   W_o[8,37] := 0.2716717;
   W_o[8,38] := -0.5921684;
   W_o[8,39] := 0.1613293;
   W_o[9,0] := -0.6345086;
   W_o[9,1] := -0.259372;
   W_o[9,2] := -0.4410478;
   W_o[9,3] := -0.1479532;
   W_o[9,4] := 0.07470662;
   W_o[9,5] := -0.1442392;
   W_o[9,6] := 0.2044672;
   W_o[9,7] := -0.3629733;
   W_o[9,8] := -0.8357224;
   W_o[9,9] := -0.03687909;
   W_o[9,10] := -0.5277801;
   W_o[9,11] := 0.1395604;
   W_o[9,12] := 0.00705423;
   W_o[9,13] := -0.06065191;
   W_o[9,14] := 0.00270301;
   W_o[9,15] := 0.02473978;
   W_o[9,16] := -0.1366292;
   W_o[9,17] := -0.1191437;
   W_o[9,18] := -0.06459489;
   W_o[9,19] := -0.155962;
   W_o[9,20] := -0.1332201;
   W_o[9,21] := 0.6168138;
   W_o[9,22] := -0.008209;
   W_o[9,23] := -0.03221058;
   W_o[9,24] := -0.07914114;
   W_o[9,25] := -0.2822376;
   W_o[9,26] := 0.1799158;
   W_o[9,27] := 0.1354283;
   W_o[9,28] := 0.1905717;
   W_o[9,29] := 0.3257442;
   W_o[9,30] := 0.2045423;
   W_o[9,31] := 0.117547;
   W_o[9,32] := 0.1869259;
   W_o[9,33] := 0.4169515;
   W_o[9,34] := 0.131826;
   W_o[9,35] := -0.1867882;
   W_o[9,36] := -0.09728058;
   W_o[9,37] := -0.2151765;
   W_o[9,38] := 0.03850761;
   W_o[9,39] := -0.0044641;
   W_o[10,0] := 0.06105608;
   W_o[10,1] := -0.06832715;
   W_o[10,2] := 0.07474305;
   W_o[10,3] := -0.08913961;
   W_o[10,4] := -0.2327598;
   W_o[10,5] := 0.07582341;
   W_o[10,6] := 0.104368;
   W_o[10,7] := 0.03688281;
   W_o[10,8] := -0.01102509;
   W_o[10,9] := -0.02805536;
   W_o[10,10] := 0.1092547;
   W_o[10,11] := -0.04491638;
   W_o[10,12] := -0.00955069;
   W_o[10,13] := -0.3600228;
   W_o[10,14] := -0.2598117;
   W_o[10,15] := -0.1312952;
   W_o[10,16] := 0.1270282;
   W_o[10,17] := 0.2455932;
   W_o[10,18] := 0.02347365;
   W_o[10,19] := 0.08953306;
   W_o[10,20] := -0.412829;
   W_o[10,21] := -0.1269261;
   W_o[10,22] := 0.1430949;
   W_o[10,23] := -0.2883692;
   W_o[10,24] := 1.613103;
   W_o[10,25] := 1.56905;
   W_o[10,26] := 0.11707;
   W_o[10,27] := -0.6253218;
   W_o[10,28] := -0.570655;
   W_o[10,29] := 0.06348585;
   W_o[10,30] := 0.2199306;
   W_o[10,31] := -0.02762064;
   W_o[10,32] := 0.08508236;
   W_o[10,33] := 0.2603731;
   W_o[10,34] := 0.5238683;
   W_o[10,35] := -0.3072915;
   W_o[10,36] := 0.4589803;
   W_o[10,37] := -0.3261147;
   W_o[10,38] := -0.04951124;
   W_o[10,39] := -0.0165583;
   W_o[11,0] := 0.2717895;
   W_o[11,1] := 0.4973186;
   W_o[11,2] := -0.111147;
   W_o[11,3] := 0.00516717;
   W_o[11,4] := -0.7287747;
   W_o[11,5] := -0.07876529;
   W_o[11,6] := -0.5072603;
   W_o[11,7] := -0.03536538;
   W_o[11,8] := 0.1201321;
   W_o[11,9] := 0.1112787;
   W_o[11,10] := 0.1532365;
   W_o[11,11] := -0.4891608;
   W_o[11,12] := 0.1887655;
   W_o[11,13] := 0.1852349;
   W_o[11,14] := 0.1703349;
   W_o[11,15] := -0.2467272;
   W_o[11,16] := 0.04845995;
   W_o[11,17] := 0.2819173;
   W_o[11,18] := 0.1057306;
   W_o[11,19] := -0.00306271;
   W_o[11,20] := -0.724054;
   W_o[11,21] := 0.09254762;
   W_o[11,22] := -0.4099866;
   W_o[11,23] := -0.1073627;
   W_o[11,24] := -0.0586772;
   W_o[11,25] := 0.3430104;
   W_o[11,26] := 0.1855343;
   W_o[11,27] := 0.1084731;
   W_o[11,28] := 0.5040212;
   W_o[11,29] := -0.00853192;
   W_o[11,30] := -0.3662441;
   W_o[11,31] := -0.01966033;
   W_o[11,32] := -0.06275205;
   W_o[11,33] := 0.09751767;
   W_o[11,34] := -0.2004695;
   W_o[11,35] := -0.1034404;
   W_o[11,36] := 0.2302412;
   W_o[11,37] := 0.1414506;
   W_o[11,38] := 0.266502;
   W_o[11,39] := -0.3097887;
   W_o[12,0] := -0.01830707;
   W_o[12,1] := 0.131161;
   W_o[12,2] := 0.00496979;
   W_o[12,3] := 0.2061931;
   W_o[12,4] := 0.03057155;
   W_o[12,5] := 0.02297443;
   W_o[12,6] := 0.05931674;
   W_o[12,7] := -0.03210922;
   W_o[12,8] := 0.07573608;
   W_o[12,9] := 0.1248056;
   W_o[12,10] := -0.07253183;
   W_o[12,11] := -0.2442229;
   W_o[12,12] := 0.1326389;
   W_o[12,13] := -0.1664325;
   W_o[12,14] := -0.1405273;
   W_o[12,15] := -0.05658006;
   W_o[12,16] := 0.04406866;
   W_o[12,17] := 0.0236842;
   W_o[12,18] := 0.7910394;
   W_o[12,19] := 0.02559086;
   W_o[12,20] := -0.1635535;
   W_o[12,21] := -0.01013497;
   W_o[12,22] := -0.3506611;
   W_o[12,23] := -0.1885774;
   W_o[12,24] := 0.4997112;
   W_o[12,25] := 0.5154855;
   W_o[12,26] := 0.1843938;
   W_o[12,27] := 0.02656424;
   W_o[12,28] := 0.00674596;
   W_o[12,29] := 0.03458697;
   W_o[12,30] := -0.4318717;
   W_o[12,31] := -0.1312484;
   W_o[12,32] := -0.3812101;
   W_o[12,33] := -0.02800291;
   W_o[12,34] := -0.2285903;
   W_o[12,35] := 0.123769;
   W_o[12,36] := 0.08067092;
   W_o[12,37] := -0.04127869;
   W_o[12,38] := -0.06010977;
   W_o[12,39] := -0.00181283;
   W_o[13,0] := -0.04045204;
   W_o[13,1] := -0.3968439;
   W_o[13,2] := 0.08165251;
   W_o[13,3] := -0.01278869;
   W_o[13,4] := -0.4479226;
   W_o[13,5] := -0.2656083;
   W_o[13,6] := 0.3235124;
   W_o[13,7] := 0.574206;
   W_o[13,8] := -0.2794143;
   W_o[13,9] := 0.3598377;
   W_o[13,10] := -0.08126416;
   W_o[13,11] := -0.00919488;
   W_o[13,12] := 0.09122144;
   W_o[13,13] := 0.02155786;
   W_o[13,14] := 0.1209246;
   W_o[13,15] := -0.00289959;
   W_o[13,16] := -0.2549352;
   W_o[13,17] := -0.2486969;
   W_o[13,18] := 0.6917394;
   W_o[13,19] := -0.03206153;
   W_o[13,20] := -0.2219304;
   W_o[13,21] := 0.1183459;
   W_o[13,22] := 0.3679306;
   W_o[13,23] := 0.4413242;
   W_o[13,24] := 1.975207;
   W_o[13,25] := 1.843769;
   W_o[13,26] := -0.279261;
   W_o[13,27] := -0.3077843;
   W_o[13,28] := -0.01960251;
   W_o[13,29] := -0.2369677;
   W_o[13,30] := 0.109645;
   W_o[13,31] := -0.1079782;
   W_o[13,32] := 0.038799;
   W_o[13,33] := 0.05485996;
   W_o[13,34] := 0.5972548;
   W_o[13,35] := 0.01886969;
   W_o[13,36] := 0.09835773;
   W_o[13,37] := 0.3843534;
   W_o[13,38] := 0.05617079;
   W_o[13,39] := -0.2227704;
   W_o[14,0] := 0.8289077;
   W_o[14,1] := -0.2031105;
   W_o[14,2] := 0.03403382;
   W_o[14,3] := 0.05452057;
   W_o[14,4] := 0.2272833;
   W_o[14,5] := -0.07046781;
   W_o[14,6] := 0.3896516;
   W_o[14,7] := 0.4871905;
   W_o[14,8] := -0.07724485;
   W_o[14,9] := -0.07247894;
   W_o[14,10] := 0.2814783;
   W_o[14,11] := -0.02350411;
   W_o[14,12] := 0.3741138;
   W_o[14,13] := 0.01457606;
   W_o[14,14] := -0.08907567;
   W_o[14,15] := 0.03109477;
   W_o[14,16] := 0.05151353;
   W_o[14,17] := -0.1566754;
   W_o[14,18] := -0.2640311;
   W_o[14,19] := -0.1076154;
   W_o[14,20] := 0.3854151;
   W_o[14,21] := 1.575822;
   W_o[14,22] := -0.05344179;
   W_o[14,23] := -0.9402446;
   W_o[14,24] := -0.0189026;
   W_o[14,25] := -0.00721721;
   W_o[14,26] := -0.4206359;
   W_o[14,27] := 0.5079048;
   W_o[14,28] := 0.2300513;
   W_o[14,29] := 0.2341685;
   W_o[14,30] := -0.1072616;
   W_o[14,31] := -0.05015407;
   W_o[14,32] := 0.03626099;
   W_o[14,33] := 0.2209553;
   W_o[14,34] := 0.2829649;
   W_o[14,35] := -0.102007;
   W_o[14,36] := 0.00415739;
   W_o[14,37] := 0.2021578;
   W_o[14,38] := 0.1449325;
   W_o[14,39] := 0.1953939;
   W_o[15,0] := 0.00236452;
   W_o[15,1] := 0.6316325;
   W_o[15,2] := 0.04516845;
   W_o[15,3] := -0.1972448;
   W_o[15,4] := -0.6675987;
   W_o[15,5] := 0.3806524;
   W_o[15,6] := 0.6475521;
   W_o[15,7] := 0.2695197;
   W_o[15,8] := -0.4985425;
   W_o[15,9] := -0.3775528;
   W_o[15,10] := 0.255392;
   W_o[15,11] := -0.1499313;
   W_o[15,12] := 0.5755351;
   W_o[15,13] := -0.03951031;
   W_o[15,14] := 0.02471058;
   W_o[15,15] := -0.2347889;
   W_o[15,16] := 0.3119133;
   W_o[15,17] := 0.02724188;
   W_o[15,18] := 0.3374691;
   W_o[15,19] := -0.0329643;
   W_o[15,20] := -0.8862573;
   W_o[15,21] := 0.5019892;
   W_o[15,22] := -0.01491885;
   W_o[15,23] := 0.393534;
   W_o[15,24] := 0.2951014;
   W_o[15,25] := 0.4423684;
   W_o[15,26] := -0.03397221;
   W_o[15,27] := -0.4513796;
   W_o[15,28] := 0.261473;
   W_o[15,29] := -0.1054694;
   W_o[15,30] := 0.3078526;
   W_o[15,31] := -0.1044204;
   W_o[15,32] := 0.2778185;
   W_o[15,33] := -0.00624027;
   W_o[15,34] := 0.2965292;
   W_o[15,35] := -0.2159247;
   W_o[15,36] := 0.05058118;
   W_o[15,37] := 0.00013962;
   W_o[15,38] := 1.000757;
   W_o[15,39] := 0.5571635;
   R_i[0,0] := -0.1137149;
   R_i[0,1] := -0.00305563;
   R_i[0,2] := 0.4498252;
   R_i[0,3] := 0.408096;
   R_i[0,4] := 0.4966823;
   R_i[0,5] := 0.2685225;
   R_i[0,6] := 0.5829936;
   R_i[0,7] := 0.309512;
   R_i[0,8] := 0.584756;
   R_i[0,9] := 0.4425567;
   R_i[0,10] := 0.168636;
   R_i[0,11] := -0.314454;
   R_i[0,12] := 0.01961905;
   R_i[0,13] := 0.3972826;
   R_i[0,14] := 0.3588874;
   R_i[0,15] := 0.1209446;
   R_i[1,0] := -0.03926941;
   R_i[1,1] := -0.2256729;
   R_i[1,2] := -0.1890858;
   R_i[1,3] := -0.4077013;
   R_i[1,4] := 1.580356;
   R_i[1,5] := -0.5334294;
   R_i[1,6] := -0.07024953;
   R_i[1,7] := 0.4276721;
   R_i[1,8] := -0.6611474;
   R_i[1,9] := 0.4677508;
   R_i[1,10] := -0.07782394;
   R_i[1,11] := -0.4426747;
   R_i[1,12] := 0.1923219;
   R_i[1,13] := 0.6306989;
   R_i[1,14] := -0.442345;
   R_i[1,15] := -0.1436543;
   R_i[2,0] := -0.1087616;
   R_i[2,1] := -0.00270978;
   R_i[2,2] := 0.2189552;
   R_i[2,3] := -0.5836519;
   R_i[2,4] := -0.07285596;
   R_i[2,5] := 0.04414057;
   R_i[2,6] := 0.2944021;
   R_i[2,7] := -0.5636789;
   R_i[2,8] := 0.02525483;
   R_i[2,9] := 0.2138523;
   R_i[2,10] := 0.1495301;
   R_i[2,11] := 0.4767698;
   R_i[2,12] := 0.3593693;
   R_i[2,13] := -0.475326;
   R_i[2,14] := -0.06119934;
   R_i[2,15] := -0.1814424;
   R_i[3,0] := -0.3477732;
   R_i[3,1] := -0.02923841;
   R_i[3,2] := -0.01545414;
   R_i[3,3] := 0.6730511;
   R_i[3,4] := 0.5243366;
   R_i[3,5] := 0.1240829;
   R_i[3,6] := 0.3667154;
   R_i[3,7] := 0.4002697;
   R_i[3,8] := 0.66468;
   R_i[3,9] := 0.1677333;
   R_i[3,10] := 0.1911234;
   R_i[3,11] := -0.5108734;
   R_i[3,12] := 0.1124746;
   R_i[3,13] := -0.2656624;
   R_i[3,14] := 0.3824491;
   R_i[3,15] := -0.1521915;
   R_i[4,0] := 0.00580328;
   R_i[4,1] := 0.6645847;
   R_i[4,2] := -0.7531157;
   R_i[4,3] := 0.00536597;
   R_i[4,4] := -1.547926;
   R_i[4,5] := -0.4703412;
   R_i[4,6] := -0.2358381;
   R_i[4,7] := 0.2062922;
   R_i[4,8] := 0.5056434;
   R_i[4,9] := 0.1705665;
   R_i[4,10] := -0.126984;
   R_i[4,11] := -1.014073;
   R_i[4,12] := 0.5201921;
   R_i[4,13] := -0.1478145;
   R_i[4,14] := -0.1872073;
   R_i[4,15] := -0.01908887;
   R_i[5,0] := -0.5724422;
   R_i[5,1] := 0.07744113;
   R_i[5,2] := 0.07027231;
   R_i[5,3] := 0.1578984;
   R_i[5,4] := 0.2315233;
   R_i[5,5] := 0.1378991;
   R_i[5,6] := -0.3647587;
   R_i[5,7] := -0.1986962;
   R_i[5,8] := -0.04011904;
   R_i[5,9] := -0.05832585;
   R_i[5,10] := -0.04800356;
   R_i[5,11] := -0.2021917;
   R_i[5,12] := -0.02367323;
   R_i[5,13] := 0.1801978;
   R_i[5,14] := 0.07786623;
   R_i[5,15] := -0.4144403;
   R_i[6,0] := -0.4898062;
   R_i[6,1] := -0.08807379;
   R_i[6,2] := 0.729624;
   R_i[6,3] := 0.5344335;
   R_i[6,4] := -0.3394561;
   R_i[6,5] := 0.02468326;
   R_i[6,6] := -0.5965754;
   R_i[6,7] := -0.1523064;
   R_i[6,8] := -0.06543954;
   R_i[6,9] := 0.0652044;
   R_i[6,10] := -0.09473334;
   R_i[6,11] := 0.06633532;
   R_i[6,12] := 0.5554917;
   R_i[6,13] := -0.5657542;
   R_i[6,14] := 0.1251685;
   R_i[6,15] := -1.210496;
   R_i[7,0] := 0.09141196;
   R_i[7,1] := -0.2953948;
   R_i[7,2] := -0.04736479;
   R_i[7,3] := 0.6381459;
   R_i[7,4] := -0.1735898;
   R_i[7,5] := 0.02200026;
   R_i[7,6] := -0.542483;
   R_i[7,7] := 0.4112348;
   R_i[7,8] := 0.08935327;
   R_i[7,9] := 0.211784;
   R_i[7,10] := 0.3778164;
   R_i[7,11] := -0.2455601;
   R_i[7,12] := -0.2529224;
   R_i[7,13] := 0.3676308;
   R_i[7,14] := -0.1642352;
   R_i[7,15] := 0.3013193;
   R_i[8,0] := -0.4359751;
   R_i[8,1] := 0.5370886;
   R_i[8,2] := -0.01918638;
   R_i[8,3] := 0.06577428;
   R_i[8,4] := -0.2360706;
   R_i[8,5] := 0.04361986;
   R_i[8,6] := 0.4372621;
   R_i[8,7] := 0.317978;
   R_i[8,8] := -1.000937;
   R_i[8,9] := -0.3358858;
   R_i[8,10] := 0.9401911;
   R_i[8,11] := -0.4844143;
   R_i[8,12] := -0.02272851;
   R_i[8,13] := 0.1828933;
   R_i[8,14] := -0.01882748;
   R_i[8,15] := -0.06172743;
   R_i[9,0] := -0.5143862;
   R_i[9,1] := 0.06295519;
   R_i[9,2] := 0.3046114;
   R_i[9,3] := 0.03788998;
   R_i[9,4] := 0.1308033;
   R_i[9,5] := -0.358474;
   R_i[9,6] := 0.69233;
   R_i[9,7] := -0.2776851;
   R_i[9,8] := 0.00155199;
   R_i[9,9] := -0.09497612;
   R_i[9,10] := 0.191216;
   R_i[9,11] := -0.428836;
   R_i[9,12] := 0.097583;
   R_i[9,13] := 0.2892125;
   R_i[9,14] := 0.1341387;
   R_i[9,15] := -0.6526389;
   R_i[10,0] := -1.243925;
   R_i[10,1] := 0.680451;
   R_i[10,2] := 0.9452817;
   R_i[10,3] := -1.115271;
   R_i[10,4] := -0.6274545;
   R_i[10,5] := -0.4702299;
   R_i[10,6] := 0.9055709;
   R_i[10,7] := 0.7863802;
   R_i[10,8] := 1.259396;
   R_i[10,9] := 0.4866133;
   R_i[10,10] := -0.232237;
   R_i[10,11] := -0.8811347;
   R_i[10,12] := -0.1416707;
   R_i[10,13] := 0.2519798;
   R_i[10,14] := 0.7145844;
   R_i[10,15] := -0.03913529;
   R_i[11,0] := -0.2986307;
   R_i[11,1] := 0.7416621;
   R_i[11,2] := -0.5418634;
   R_i[11,3] := -0.0208676;
   R_i[11,4] := 0.4454969;
   R_i[11,5] := -0.1592286;
   R_i[11,6] := 0.2505509;
   R_i[11,7] := -0.382692;
   R_i[11,8] := 0.1618413;
   R_i[11,9] := 0.4193928;
   R_i[11,10] := 0.02712804;
   R_i[11,11] := -1.186852;
   R_i[11,12] := 0.2001949;
   R_i[11,13] := 0.1532502;
   R_i[11,14] := -0.3284004;
   R_i[11,15] := -0.2820552;
   R_i[12,0] := -0.2895075;
   R_i[12,1] := 1.091435;
   R_i[12,2] := -0.05338987;
   R_i[12,3] := 0.2911161;
   R_i[12,4] := 0.1629717;
   R_i[12,5] := -0.161591;
   R_i[12,6] := 0.5146877;
   R_i[12,7] := 0.03626299;
   R_i[12,8] := 0.08357667;
   R_i[12,9] := 0.2767582;
   R_i[12,10] := -0.2725959;
   R_i[12,11] := -0.9445232;
   R_i[12,12] := 2.164176;
   R_i[12,13] := -0.04564672;
   R_i[12,14] := -0.9437686;
   R_i[12,15] := -0.3752556;
   R_i[13,0] := -0.3738814;
   R_i[13,1] := -0.4302073;
   R_i[13,2] := 0.06173271;
   R_i[13,3] := -0.3280604;
   R_i[13,4] := -0.2716264;
   R_i[13,5] := 0.3550667;
   R_i[13,6] := -0.05685175;
   R_i[13,7] := 0.5135436;
   R_i[13,8] := 0.1640313;
   R_i[13,9] := -0.2691319;
   R_i[13,10] := -0.3801848;
   R_i[13,11] := 0.1228051;
   R_i[13,12] := 0.5428029;
   R_i[13,13] := 1.709359;
   R_i[13,14] := 1.011569;
   R_i[13,15] := -0.4288203;
   R_i[14,0] := 0.2300761;
   R_i[14,1] := -1.012092;
   R_i[14,2] := 0.6361403;
   R_i[14,3] := 0.05786986;
   R_i[14,4] := -0.4553789;
   R_i[14,5] := -0.6679262;
   R_i[14,6] := -0.4034081;
   R_i[14,7] := 0.00973069;
   R_i[14,8] := 1.011842;
   R_i[14,9] := -0.3590509;
   R_i[14,10] := 0.3335861;
   R_i[14,11] := -0.8217174;
   R_i[14,12] := -0.6475059;
   R_i[14,13] := -0.2020338;
   R_i[14,14] := 3.036138;
   R_i[14,15] := -0.1744984;
   R_i[15,0] := -0.04125203;
   R_i[15,1] := 0.6700256;
   R_i[15,2] := 1.07735;
   R_i[15,3] := 0.2874972;
   R_i[15,4] := -0.03804383;
   R_i[15,5] := 0.0777116;
   R_i[15,6] := 0.6422315;
   R_i[15,7] := 0.2854839;
   R_i[15,8] := 0.2419276;
   R_i[15,9] := 0.0058566;
   R_i[15,10] := 0.6288991;
   R_i[15,11] := -0.8346034;
   R_i[15,12] := 0.2495139;
   R_i[15,13] := -0.4616964;
   R_i[15,14] := 0.8547717;
   R_i[15,15] := -1.059702;
   R_f[0,0] := 0.3233714;
   R_f[0,1] := -0.6415426;
   R_f[0,2] := 0.4436696;
   R_f[0,3] := -0.1691184;
   R_f[0,4] := -0.2260693;
   R_f[0,5] := 0.4070715;
   R_f[0,6] := 0.9958715;
   R_f[0,7] := -0.6152283;
   R_f[0,8] := -0.1669062;
   R_f[0,9] := 0.1140058;
   R_f[0,10] := -1.301264;
   R_f[0,11] := 0.6843588;
   R_f[0,12] := 0.2550505;
   R_f[0,13] := -0.5000576;
   R_f[0,14] := 1.899208;
   R_f[0,15] := 0.3119706;
   R_f[1,0] := -0.1011617;
   R_f[1,1] := 3.477333;
   R_f[1,2] := -0.2395845;
   R_f[1,3] := 0.2576158;
   R_f[1,4] := 0.6485823;
   R_f[1,5] := 0.2552066;
   R_f[1,6] := 0.4734288;
   R_f[1,7] := 0.4439468;
   R_f[1,8] := 0.08832169;
   R_f[1,9] := -0.07672439;
   R_f[1,10] := -0.1136505;
   R_f[1,11] := -0.1276775;
   R_f[1,12] := 0.153016;
   R_f[1,13] := 0.1081575;
   R_f[1,14] := -0.00451868;
   R_f[1,15] := 0.1695628;
   R_f[2,0] := 0.8806943;
   R_f[2,1] := -0.4307577;
   R_f[2,2] := -0.285418;
   R_f[2,3] := 0.7795734;
   R_f[2,4] := 0.49964;
   R_f[2,5] := 0.1542652;
   R_f[2,6] := 0.2286351;
   R_f[2,7] := -0.7402638;
   R_f[2,8] := -0.6850481;
   R_f[2,9] := -0.3444061;
   R_f[2,10] := -0.5146202;
   R_f[2,11] := 0.5203135;
   R_f[2,12] := -0.2921089;
   R_f[2,13] := -0.7581262;
   R_f[2,14] := 0.2400508;
   R_f[2,15] := 0.06470054;
   R_f[3,0] := -1.016384;
   R_f[3,1] := -0.01572494;
   R_f[3,2] := 1.122687;
   R_f[3,3] := -1.076523;
   R_f[3,4] := -0.2219028;
   R_f[3,5] := 0.3841916;
   R_f[3,6] := 0.6512823;
   R_f[3,7] := 1.68439;
   R_f[3,8] := 0.7787917;
   R_f[3,9] := -0.1303423;
   R_f[3,10] := 0.1025792;
   R_f[3,11] := 0.0630113;
   R_f[3,12] := -0.2613996;
   R_f[3,13] := 0.08574831;
   R_f[3,14] := 0.5817915;
   R_f[3,15] := -0.1694773;
   R_f[4,0] := -0.09817147;
   R_f[4,1] := -0.8673013;
   R_f[4,2] := 0.1123603;
   R_f[4,3] := -0.05304767;
   R_f[4,4] := -0.1617602;
   R_f[4,5] := -0.4315653;
   R_f[4,6] := -0.1545042;
   R_f[4,7] := -0.04651795;
   R_f[4,8] := -0.7793221;
   R_f[4,9] := 0.2078234;
   R_f[4,10] := 0.1676973;
   R_f[4,11] := 0.3325663;
   R_f[4,12] := 0.157971;
   R_f[4,13] := 0.7362291;
   R_f[4,14] := 0.0176266;
   R_f[4,15] := -0.6734453;
   R_f[5,0] := 1.169603;
   R_f[5,1] := -0.73158;
   R_f[5,2] := 0.4122632;
   R_f[5,3] := 0.02196453;
   R_f[5,4] := 0.3548708;
   R_f[5,5] := 0.1889586;
   R_f[5,6] := 0.3045126;
   R_f[5,7] := 0.9211732;
   R_f[5,8] := -0.4857724;
   R_f[5,9] := -0.9820208;
   R_f[5,10] := -0.5130315;
   R_f[5,11] := 0.2623543;
   R_f[5,12] := -0.2203466;
   R_f[5,13] := -1.837646;
   R_f[5,14] := -0.6587409;
   R_f[5,15] := -0.2930804;
   R_f[6,0] := -0.3989139;
   R_f[6,1] := -0.7530556;
   R_f[6,2] := 1.695848;
   R_f[6,3] := -0.1637086;
   R_f[6,4] := 0.2540572;
   R_f[6,5] := 0.02853256;
   R_f[6,6] := 0.1514727;
   R_f[6,7] := -1.134142;
   R_f[6,8] := -0.9914478;
   R_f[6,9] := -0.4490964;
   R_f[6,10] := -0.6475779;
   R_f[6,11] := -0.02062916;
   R_f[6,12] := 0.3351462;
   R_f[6,13] := 0.3090186;
   R_f[6,14] := 0.6139765;
   R_f[6,15] := 0.7687923;
   R_f[7,0] := -0.2705219;
   R_f[7,1] := 0.04162847;
   R_f[7,2] := 3.147241;
   R_f[7,3] := -0.331195;
   R_f[7,4] := -0.5884408;
   R_f[7,5] := -0.3636526;
   R_f[7,6] := -0.9163497;
   R_f[7,7] := 0.3539489;
   R_f[7,8] := 0.2825061;
   R_f[7,9] := 0.493275;
   R_f[7,10] := 1.353475;
   R_f[7,11] := -1.124487;
   R_f[7,12] := -0.5918967;
   R_f[7,13] := 1.290014;
   R_f[7,14] := -0.550961;
   R_f[7,15] := 0.8665411;
   R_f[8,0] := 0.3655965;
   R_f[8,1] := -1.387398;
   R_f[8,2] := 0.6403066;
   R_f[8,3] := 0.4521842;
   R_f[8,4] := 0.426568;
   R_f[8,5] := -0.3468258;
   R_f[8,6] := -1.100012;
   R_f[8,7] := -0.6693547;
   R_f[8,8] := -3.069017;
   R_f[8,9] := 0.1657671;
   R_f[8,10] := 0.784942;
   R_f[8,11] := -0.4345917;
   R_f[8,12] := -1.434882;
   R_f[8,13] := 0.1338141;
   R_f[8,14] := -0.793483;
   R_f[8,15] := -0.2249214;
   R_f[9,0] := -0.152597;
   R_f[9,1] := -1.499914;
   R_f[9,2] := 1.108761;
   R_f[9,3] := -0.5297781;
   R_f[9,4] := -0.6886869;
   R_f[9,5] := -1.672909;
   R_f[9,6] := 2.633435;
   R_f[9,7] := -1.828544;
   R_f[9,8] := -0.740662;
   R_f[9,9] := 1.526205;
   R_f[9,10] := 0.4746018;
   R_f[9,11] := 1.381489;
   R_f[9,12] := -0.6054185;
   R_f[9,13] := 0.7926679;
   R_f[9,14] := 0.3271781;
   R_f[9,15] := -1.000112;
   R_f[10,0] := 2.164407;
   R_f[10,1] := -0.6995372;
   R_f[10,2] := 0.6653332;
   R_f[10,3] := 1.181759;
   R_f[10,4] := -0.2965346;
   R_f[10,5] := -0.1037577;
   R_f[10,6] := 0.02757812;
   R_f[10,7] := -0.9681873;
   R_f[10,8] := -0.4607585;
   R_f[10,9] := -0.5446746;
   R_f[10,10] := 0.780597;
   R_f[10,11] := -0.7688502;
   R_f[10,12] := -1.056067;
   R_f[10,13] := -0.1988855;
   R_f[10,14] := 0.01456859;
   R_f[10,15] := 0.3702135;
   R_f[11,0] := 0.2434937;
   R_f[11,1] := -0.1798942;
   R_f[11,2] := 0.2355876;
   R_f[11,3] := -0.6682997;
   R_f[11,4] := -0.5007147;
   R_f[11,5] := -0.5791205;
   R_f[11,6] := 0.1253008;
   R_f[11,7] := -0.7620748;
   R_f[11,8] := -0.5787513;
   R_f[11,9] := 0.0264844;
   R_f[11,10] := 0.4317927;
   R_f[11,11] := -1.222577;
   R_f[11,12] := -0.03755289;
   R_f[11,13] := -0.1228497;
   R_f[11,14] := 0.0646783;
   R_f[11,15] := 0.2649987;
   R_f[12,0] := -0.02412502;
   R_f[12,1] := -0.4178893;
   R_f[12,2] := 0.2250565;
   R_f[12,3] := 0.2468531;
   R_f[12,4] := -0.2603359;
   R_f[12,5] := 0.5588626;
   R_f[12,6] := 0.3501927;
   R_f[12,7] := 0.0646469;
   R_f[12,8] := 0.3895332;
   R_f[12,9] := 0.409056;
   R_f[12,10] := 0.161415;
   R_f[12,11] := -0.05112006;
   R_f[12,12] := 1.493768;
   R_f[12,13] := 0.3131461;
   R_f[12,14] := 0.4573432;
   R_f[12,15] := 0.3800302;
   R_f[13,0] := 0.5914586;
   R_f[13,1] := -0.351166;
   R_f[13,2] := 0.8291268;
   R_f[13,3] := 0.2013447;
   R_f[13,4] := 0.82876;
   R_f[13,5] := 0.8977232;
   R_f[13,6] := 1.657781;
   R_f[13,7] := 0.4952854;
   R_f[13,8] := -0.8510268;
   R_f[13,9] := -0.7816306;
   R_f[13,10] := 0.3712052;
   R_f[13,11] := 0.7794952;
   R_f[13,12] := -0.1510022;
   R_f[13,13] := -0.1749281;
   R_f[13,14] := -0.00674355;
   R_f[13,15] := -0.6594451;
   R_f[14,0] := -0.03948923;
   R_f[14,1] := -0.3682528;
   R_f[14,2] := 1.244398;
   R_f[14,3] := -0.5374001;
   R_f[14,4] := -0.4286888;
   R_f[14,5] := 0.2608948;
   R_f[14,6] := 0.4886785;
   R_f[14,7] := 1.195282;
   R_f[14,8] := 0.1545673;
   R_f[14,9] := -1.140402;
   R_f[14,10] := 0.05182516;
   R_f[14,11] := -0.2172662;
   R_f[14,12] := 0.1702152;
   R_f[14,13] := -0.6474801;
   R_f[14,14] := 1.387721;
   R_f[14,15] := 0.2322865;
   R_f[15,0] := 0.3153065;
   R_f[15,1] := -0.9808237;
   R_f[15,2] := 0.2264991;
   R_f[15,3] := -0.2976737;
   R_f[15,4] := 0.5468484;
   R_f[15,5] := 0.7780918;
   R_f[15,6] := 2.003952;
   R_f[15,7] := 2.355743;
   R_f[15,8] := -0.1702361;
   R_f[15,9] := -0.381211;
   R_f[15,10] := 1.069254;
   R_f[15,11] := -0.3054578;
   R_f[15,12] := -0.4347287;
   R_f[15,13] := -1.114827;
   R_f[15,14] := 0.3245434;
   R_f[15,15] := -1.337709;
   R_g[0,0] := -2.805433;
   R_g[0,1] := 0.09675837;
   R_g[0,2] := 0.04763355;
   R_g[0,3] := 0.1613498;
   R_g[0,4] := -0.04916951;
   R_g[0,5] := 0.06786807;
   R_g[0,6] := 0.07195669;
   R_g[0,7] := 0.1879627;
   R_g[0,8] := 0.02096096;
   R_g[0,9] := -0.05091592;
   R_g[0,10] := 0.1711352;
   R_g[0,11] := 0.09710391;
   R_g[0,12] := -0.1928508;
   R_g[0,13] := 0.04608029;
   R_g[0,14] := 0.3775772;
   R_g[0,15] := -0.05004899;
   R_g[1,0] := 0.08712953;
   R_g[1,1] := -1.281738;
   R_g[1,2] := 0.486291;
   R_g[1,3] := -0.1018547;
   R_g[1,4] := 0.5911466;
   R_g[1,5] := 0.3826247;
   R_g[1,6] := 0.04029783;
   R_g[1,7] := 0.06582787;
   R_g[1,8] := -0.06752597;
   R_g[1,9] := -0.2294858;
   R_g[1,10] := -0.1253151;
   R_g[1,11] := -0.2067355;
   R_g[1,12] := -0.05208173;
   R_g[1,13] := 0.1810765;
   R_g[1,14] := 0.05905702;
   R_g[1,15] := -0.06634986;
   R_g[2,0] := -0.2549139;
   R_g[2,1] := -0.05303259;
   R_g[2,2] := -3.258265;
   R_g[2,3] := 0.2239036;
   R_g[2,4] := 0.08010214;
   R_g[2,5] := 0.1251935;
   R_g[2,6] := -0.1281362;
   R_g[2,7] := 0.03709217;
   R_g[2,8] := -0.0533942;
   R_g[2,9] := -0.1838315;
   R_g[2,10] := 0.01583981;
   R_g[2,11] := 0.1206139;
   R_g[2,12] := 0.02361463;
   R_g[2,13] := 0.1162473;
   R_g[2,14] := 0.1685608;
   R_g[2,15] := -0.04670952;
   R_g[3,0] := -0.3499806;
   R_g[3,1] := 0.7145555;
   R_g[3,2] := -0.7979932;
   R_g[3,3] := -2.84151;
   R_g[3,4] := 0.1580465;
   R_g[3,5] := -0.08033045;
   R_g[3,6] := -0.1452473;
   R_g[3,7] := 0.2225952;
   R_g[3,8] := 0.07427457;
   R_g[3,9] := 0.3725025;
   R_g[3,10] := -0.308892;
   R_g[3,11] := -0.2322429;
   R_g[3,12] := 0.6733903;
   R_g[3,13] := 0.1802014;
   R_g[3,14] := -0.04057474;
   R_g[3,15] := -0.1780594;
   R_g[4,0] := 0.4558564;
   R_g[4,1] := 0.2691017;
   R_g[4,2] := 0.2479934;
   R_g[4,3] := 0.1830495;
   R_g[4,4] := -2.643592;
   R_g[4,5] := -0.1854873;
   R_g[4,6] := 0.5796254;
   R_g[4,7] := -0.2360368;
   R_g[4,8] := 0.3996172;
   R_g[4,9] := -0.08552616;
   R_g[4,10] := -0.3547961;
   R_g[4,11] := 0.02176627;
   R_g[4,12] := -0.1695444;
   R_g[4,13] := -0.6054811;
   R_g[4,14] := 0.05480947;
   R_g[4,15] := 0.2614591;
   R_g[5,0] := 0.09851117;
   R_g[5,1] := 0.05978253;
   R_g[5,2] := -0.2238024;
   R_g[5,3] := 0.06287329;
   R_g[5,4] := 0.2952785;
   R_g[5,5] := -6.417284;
   R_g[5,6] := -0.01966351;
   R_g[5,7] := 0.08289347;
   R_g[5,8] := 0.2335418;
   R_g[5,9] := 0.4640638;
   R_g[5,10] := -0.5190796;
   R_g[5,11] := -0.3999299;
   R_g[5,12] := 0.3029557;
   R_g[5,13] := 0.06150499;
   R_g[5,14] := -1.054952;
   R_g[5,15] := -0.08431676;
   R_g[6,0] := -0.1025641;
   R_g[6,1] := 0.05051776;
   R_g[6,2] := 0.0306027;
   R_g[6,3] := 0.06608646;
   R_g[6,4] := -0.05028161;
   R_g[6,5] := -0.1038706;
   R_g[6,6] := -3.13754;
   R_g[6,7] := -0.1565541;
   R_g[6,8] := 0.03909466;
   R_g[6,9] := -0.03506904;
   R_g[6,10] := 0.0048442;
   R_g[6,11] := -0.1906409;
   R_g[6,12] := 0.330723;
   R_g[6,13] := -0.06755624;
   R_g[6,14] := -0.1569814;
   R_g[6,15] := -0.3220711;
   R_g[7,0] := 0.07863971;
   R_g[7,1] := -0.1875482;
   R_g[7,2] := -0.2537812;
   R_g[7,3] := -0.08824939;
   R_g[7,4] := -0.1294116;
   R_g[7,5] := 0.2885412;
   R_g[7,6] := 0.1121606;
   R_g[7,7] := -3.136752;
   R_g[7,8] := -0.08472223;
   R_g[7,9] := 0.00790842;
   R_g[7,10] := -0.1138648;
   R_g[7,11] := -0.05684523;
   R_g[7,12] := 0.1106585;
   R_g[7,13] := -0.07569506;
   R_g[7,14] := 0.4233017;
   R_g[7,15] := -0.1342552;
   R_g[8,0] := 0.08961181;
   R_g[8,1] := 0.4651947;
   R_g[8,2] := -0.3656231;
   R_g[8,3] := 0.2111352;
   R_g[8,4] := -0.00757714;
   R_g[8,5] := -0.2639286;
   R_g[8,6] := 0.1638752;
   R_g[8,7] := -0.4058702;
   R_g[8,8] := -2.934379;
   R_g[8,9] := 0.08376594;
   R_g[8,10] := -0.2960652;
   R_g[8,11] := 0.01828978;
   R_g[8,12] := 0.2524873;
   R_g[8,13] := -0.3134462;
   R_g[8,14] := -0.01567479;
   R_g[8,15] := 0.05443858;
   R_g[9,0] := -0.1509652;
   R_g[9,1] := -0.2985869;
   R_g[9,2] := 0.1976654;
   R_g[9,3] := -0.1125526;
   R_g[9,4] := -0.1207261;
   R_g[9,5] := 0.337102;
   R_g[9,6] := 0.2015858;
   R_g[9,7] := -0.1138979;
   R_g[9,8] := -0.08645659;
   R_g[9,9] := -4.490891;
   R_g[9,10] := 0.03153508;
   R_g[9,11] := 0.1759175;
   R_g[9,12] := -0.00816477;
   R_g[9,13] := -0.09244221;
   R_g[9,14] := -0.1702342;
   R_g[9,15] := 0.4290646;
   R_g[10,0] := -0.3885716;
   R_g[10,1] := 0.0643687;
   R_g[10,2] := -0.1564249;
   R_g[10,3] := -0.1040558;
   R_g[10,4] := 0.1323418;
   R_g[10,5] := 0.1366159;
   R_g[10,6] := 0.04957649;
   R_g[10,7] := 0.0648922;
   R_g[10,8] := 0.1469345;
   R_g[10,9] := -0.01300282;
   R_g[10,10] := -1.928301;
   R_g[10,11] := 0.3004588;
   R_g[10,12] := 0.2731377;
   R_g[10,13] := 0.02955168;
   R_g[10,14] := -0.07842075;
   R_g[10,15] := 0.05753986;
   R_g[11,0] := -0.2097152;
   R_g[11,1] := 0.7307096;
   R_g[11,2] := -0.503158;
   R_g[11,3] := 0.205001;
   R_g[11,4] := -0.01089373;
   R_g[11,5] := 0.16405;
   R_g[11,6] := 0.1890694;
   R_g[11,7] := 0.03491729;
   R_g[11,8] := -0.01610962;
   R_g[11,9] := 0.2807466;
   R_g[11,10] := 0.02013272;
   R_g[11,11] := -4.203784;
   R_g[11,12] := 0.2934183;
   R_g[11,13] := 0.1436955;
   R_g[11,14] := -0.41985;
   R_g[11,15] := 0.0576296;
   R_g[12,0] := -0.03705381;
   R_g[12,1] := -0.3112487;
   R_g[12,2] := 0.6347389;
   R_g[12,3] := 0.08633271;
   R_g[12,4] := -0.1792604;
   R_g[12,5] := 0.317774;
   R_g[12,6] := -0.1986456;
   R_g[12,7] := -0.1977208;
   R_g[12,8] := 0.1422061;
   R_g[12,9] := -0.2642545;
   R_g[12,10] := 0.07095157;
   R_g[12,11] := 0.5123266;
   R_g[12,12] := -3.63069;
   R_g[12,13] := -0.1175799;
   R_g[12,14] := 0.2990645;
   R_g[12,15] := -0.02980175;
   R_g[13,0] := 0.00863379;
   R_g[13,1] := 0.03295338;
   R_g[13,2] := -0.3002235;
   R_g[13,3] := 0.1032756;
   R_g[13,4] := -0.1160595;
   R_g[13,5] := 0.031227;
   R_g[13,6] := 0.6257741;
   R_g[13,7] := 0.4343066;
   R_g[13,8] := 0.1252338;
   R_g[13,9] := 0.1524162;
   R_g[13,10] := -0.2399488;
   R_g[13,11] := -0.0243434;
   R_g[13,12] := 0.07577311;
   R_g[13,13] := -2.642776;
   R_g[13,14] := -0.7371749;
   R_g[13,15] := -0.08735505;
   R_g[14,0] := -0.171414;
   R_g[14,1] := 0.2261713;
   R_g[14,2] := -0.3317359;
   R_g[14,3] := 0.0877693;
   R_g[14,4] := 0.1621639;
   R_g[14,5] := 0.2182705;
   R_g[14,6] := 0.04451356;
   R_g[14,7] := 0.03265934;
   R_g[14,8] := -0.136193;
   R_g[14,9] := 0.1847814;
   R_g[14,10] := -0.0108934;
   R_g[14,11] := -0.2341314;
   R_g[14,12] := 0.1122679;
   R_g[14,13] := 0.2223738;
   R_g[14,14] := -2.0286;
   R_g[14,15] := -0.01800863;
   R_g[15,0] := 0.3883483;
   R_g[15,1] := -0.1211964;
   R_g[15,2] := -0.4713392;
   R_g[15,3] := 0.02589257;
   R_g[15,4] := -0.1296599;
   R_g[15,5] := -0.2871422;
   R_g[15,6] := 0.6408823;
   R_g[15,7] := 0.4650818;
   R_g[15,8] := -0.1301513;
   R_g[15,9] := 0.1214571;
   R_g[15,10] := 0.3844216;
   R_g[15,11] := -0.5117303;
   R_g[15,12] := -0.03178278;
   R_g[15,13] := -0.2080431;
   R_g[15,14] := 0.6247337;
   R_g[15,15] := -3.379229;
   R_o[0,0] := -0.148473;
   R_o[0,1] := -0.7470531;
   R_o[0,2] := 0.337931;
   R_o[0,3] := 0.4881276;
   R_o[0,4] := -0.5424621;
   R_o[0,5] := 0.2365883;
   R_o[0,6] := 0.3687733;
   R_o[0,7] := -0.04479291;
   R_o[0,8] := 0.04525228;
   R_o[0,9] := -0.06947453;
   R_o[0,10] := -0.2940823;
   R_o[0,11] := -0.6614071;
   R_o[0,12] := -0.09016941;
   R_o[0,13] := -0.2445324;
   R_o[0,14] := 0.4173301;
   R_o[0,15] := 0.1152808;
   R_o[1,0] := -0.2253625;
   R_o[1,1] := -2.687598;
   R_o[1,2] := 0.7825195;
   R_o[1,3] := 0.3311445;
   R_o[1,4] := -0.6487191;
   R_o[1,5] := -0.1774464;
   R_o[1,6] := -0.6072173;
   R_o[1,7] := -0.9984445;
   R_o[1,8] := 0.693763;
   R_o[1,9] := -0.04945409;
   R_o[1,10] := 0.1380522;
   R_o[1,11] := 0.2601311;
   R_o[1,12] := -0.5988305;
   R_o[1,13] := -1.649512;
   R_o[1,14] := -0.06540374;
   R_o[1,15] := -0.683998;
   R_o[2,0] := 0.1426505;
   R_o[2,1] := -0.7636122;
   R_o[2,2] := 0.6522185;
   R_o[2,3] := -0.01308598;
   R_o[2,4] := -0.3956572;
   R_o[2,5] := -0.1286385;
   R_o[2,6] := 0.1117783;
   R_o[2,7] := -0.1965184;
   R_o[2,8] := 0.445568;
   R_o[2,9] := -0.3197942;
   R_o[2,10] := 0.1024574;
   R_o[2,11] := -0.3961471;
   R_o[2,12] := -0.1107483;
   R_o[2,13] := -0.7957024;
   R_o[2,14] := 0.2206428;
   R_o[2,15] := 0.2849079;
   R_o[3,0] := 0.103478;
   R_o[3,1] := -0.3351506;
   R_o[3,2] := 0.1007192;
   R_o[3,3] := 0.2476437;
   R_o[3,4] := -0.3063624;
   R_o[3,5] := -0.02347863;
   R_o[3,6] := 0.6147529;
   R_o[3,7] := 0.05460903;
   R_o[3,8] := -0.09153262;
   R_o[3,9] := -0.07667586;
   R_o[3,10] := 0.1709715;
   R_o[3,11] := -0.847174;
   R_o[3,12] := 0.01488861;
   R_o[3,13] := 0.01246201;
   R_o[3,14] := 0.785248;
   R_o[3,15] := -0.2429155;
   R_o[4,0] := 0.7403428;
   R_o[4,1] := -1.202408;
   R_o[4,2] := -0.01728833;
   R_o[4,3] := -0.2675001;
   R_o[4,4] := 0.4232838;
   R_o[4,5] := -0.1884229;
   R_o[4,6] := -0.4024306;
   R_o[4,7] := 0.6314479;
   R_o[4,8] := -1.543486;
   R_o[4,9] := 0.5625891;
   R_o[4,10] := -0.4602357;
   R_o[4,11] := -0.7463102;
   R_o[4,12] := 0.01794407;
   R_o[4,13] := 0.6175683;
   R_o[4,14] := -0.4240062;
   R_o[4,15] := -0.3216551;
   R_o[5,0] := -1.608714;
   R_o[5,1] := -0.8543944;
   R_o[5,2] := 0.1236723;
   R_o[5,3] := 0.3216394;
   R_o[5,4] := -0.4782757;
   R_o[5,5] := 3.932515;
   R_o[5,6] := -0.1368901;
   R_o[5,7] := 1.26777;
   R_o[5,8] := -0.6972287;
   R_o[5,9] := -0.6138417;
   R_o[5,10] := 0.9199839;
   R_o[5,11] := -0.644981;
   R_o[5,12] := -0.2947383;
   R_o[5,13] := -1.30751;
   R_o[5,14] := 0.8453699;
   R_o[5,15] := 1.6406;
   R_o[6,0] := 0.02413699;
   R_o[6,1] := -0.7911229;
   R_o[6,2] := -0.1035878;
   R_o[6,3] := -0.345346;
   R_o[6,4] := 0.4822478;
   R_o[6,5] := -0.5942275;
   R_o[6,6] := 0.5900132;
   R_o[6,7] := 0.05578557;
   R_o[6,8] := -0.1626476;
   R_o[6,9] := -0.5127108;
   R_o[6,10] := 0.395417;
   R_o[6,11] := -0.5891114;
   R_o[6,12] := -0.04537732;
   R_o[6,13] := 0.2378311;
   R_o[6,14] := 0.5396131;
   R_o[6,15] := 0.6403692;
   R_o[7,0] := 0.1401259;
   R_o[7,1] := -1.107673;
   R_o[7,2] := 0.449949;
   R_o[7,3] := 0.1980791;
   R_o[7,4] := -0.1763375;
   R_o[7,5] := -0.02624386;
   R_o[7,6] := 0.6654956;
   R_o[7,7] := 0.8419639;
   R_o[7,8] := 0.07700922;
   R_o[7,9] := 0.585766;
   R_o[7,10] := 0.117281;
   R_o[7,11] := -0.205901;
   R_o[7,12] := -0.1026604;
   R_o[7,13] := 0.1098014;
   R_o[7,14] := 0.8365094;
   R_o[7,15] := 0.4066797;
   R_o[8,0] := 0.1040777;
   R_o[8,1] := -1.388284;
   R_o[8,2] := 0.5748492;
   R_o[8,3] := -0.3209612;
   R_o[8,4] := -1.21653;
   R_o[8,5] := -0.1644516;
   R_o[8,6] := 0.521858;
   R_o[8,7] := 2.041153;
   R_o[8,8] := -2.922855;
   R_o[8,9] := -0.6003711;
   R_o[8,10] := -0.1361148;
   R_o[8,11] := -0.102449;
   R_o[8,12] := -0.5256941;
   R_o[8,13] := -0.3414919;
   R_o[8,14] := 0.9229004;
   R_o[8,15] := -0.1494768;
   R_o[9,0] := 0.9020318;
   R_o[9,1] := -1.182273;
   R_o[9,2] := 0.7037838;
   R_o[9,3] := -0.07063206;
   R_o[9,4] := -0.4500138;
   R_o[9,5] := 0.3359483;
   R_o[9,6] := 0.9089686;
   R_o[9,7] := -0.1131394;
   R_o[9,8] := 0.06154737;
   R_o[9,9] := -3.070117;
   R_o[9,10] := 0.2449786;
   R_o[9,11] := -0.03553757;
   R_o[9,12] := -0.3328317;
   R_o[9,13] := 0.3393808;
   R_o[9,14] := 0.4877961;
   R_o[9,15] := 0.9906611;
   R_o[10,0] := 0.3674809;
   R_o[10,1] := -0.4065204;
   R_o[10,2] := 0.3212383;
   R_o[10,3] := 0.1469396;
   R_o[10,4] := -0.8636696;
   R_o[10,5] := 0.4387633;
   R_o[10,6] := -0.3679813;
   R_o[10,7] := -0.3709672;
   R_o[10,8] := 0.8587736;
   R_o[10,9] := -0.4086122;
   R_o[10,10] := 1.240259;
   R_o[10,11] := -0.5606848;
   R_o[10,12] := -0.1593753;
   R_o[10,13] := -0.5910825;
   R_o[10,14] := 0.8222155;
   R_o[10,15] := 0.07025416;
   R_o[11,0] := -0.283336;
   R_o[11,1] := -0.8366182;
   R_o[11,2] := 0.2441355;
   R_o[11,3] := 0.1767131;
   R_o[11,4] := -0.4013823;
   R_o[11,5] := 0.1624961;
   R_o[11,6] := 0.590718;
   R_o[11,7] := 1.182436;
   R_o[11,8] := -0.1144639;
   R_o[11,9] := -0.459346;
   R_o[11,10] := 0.4479548;
   R_o[11,11] := 1.724371;
   R_o[11,12] := -0.6445624;
   R_o[11,13] := -0.2646877;
   R_o[11,14] := 1.049319;
   R_o[11,15] := 1.146086;
   R_o[12,0] := 0.06811738;
   R_o[12,1] := -0.8294082;
   R_o[12,2] := 0.04298686;
   R_o[12,3] := 0.1884655;
   R_o[12,4] := -0.4888053;
   R_o[12,5] := 0.06246455;
   R_o[12,6] := 0.5130124;
   R_o[12,7] := 0.01585177;
   R_o[12,8] := -0.3286436;
   R_o[12,9] := -0.1914053;
   R_o[12,10] := 0.3550029;
   R_o[12,11] := -0.6732444;
   R_o[12,12] := -0.1367572;
   R_o[12,13] := 0.1686232;
   R_o[12,14] := 0.7652449;
   R_o[12,15] := 0.1804299;
   R_o[13,0] := 1.529198;
   R_o[13,1] := -2.016652;
   R_o[13,2] := 0.07069629;
   R_o[13,3] := 0.5932482;
   R_o[13,4] := -0.01248456;
   R_o[13,5] := 0.1003619;
   R_o[13,6] := 0.9069089;
   R_o[13,7] := 0.4181206;
   R_o[13,8] := -0.1110177;
   R_o[13,9] := -0.4146234;
   R_o[13,10] := 0.3274502;
   R_o[13,11] := 0.09499595;
   R_o[13,12] := -1.174091;
   R_o[13,13] := 0.9226585;
   R_o[13,14] := 0.3798864;
   R_o[13,15] := 0.05125737;
   R_o[14,0] := 4.215199;
   R_o[14,1] := -0.6910225;
   R_o[14,2] := 0.0060396;
   R_o[14,3] := -2.409633;
   R_o[14,4] := -0.6553826;
   R_o[14,5] := -0.06152564;
   R_o[14,6] := -1.545334;
   R_o[14,7] := -0.2254379;
   R_o[14,8] := 1.58575;
   R_o[14,9] := -0.1091707;
   R_o[14,10] := 1.547734;
   R_o[14,11] := -0.1732163;
   R_o[14,12] := -0.8589516;
   R_o[14,13] := -1.472137;
   R_o[14,14] := 2.376655;
   R_o[14,15] := -1.796365;
   R_o[15,0] := 1.089969;
   R_o[15,1] := -1.172117;
   R_o[15,2] := 0.6316615;
   R_o[15,3] := 0.516769;
   R_o[15,4] := -0.3734112;
   R_o[15,5] := 0.6013339;
   R_o[15,6] := 1.511744;
   R_o[15,7] := 0.264806;
   R_o[15,8] := 0.3243769;
   R_o[15,9] := -0.585372;
   R_o[15,10] := -0.03915246;
   R_o[15,11] := -0.1954393;
   R_o[15,12] := -0.8276399;
   R_o[15,13] := 0.3127334;
   R_o[15,14] := 0.7691328;
   R_o[15,15] := 0.7349373;
   B_i[0] := -0.1152518;
   B_i[1] := -0.1676714;
   B_i[2] := -0.1067528;
   B_i[3] := 0.275955;
   B_i[4] := 0.1112795;
   B_i[5] := -1.207003;
   B_i[6] := -0.3355503;
   B_i[7] := -0.3521997;
   B_i[8] := -0.03516939;
   B_i[9] := -0.6599523;
   B_i[10] := 1.630978;
   B_i[11] := -0.183339;
   B_i[12] := 0.07472892;
   B_i[13] := 0.2571971;
   B_i[14] := -0.1915112;
   B_i[15] := -0.6759596;
   B_f[0] := 2.995566;
   B_f[1] := -0.337418;
   B_f[2] := 2.251579;
   B_f[3] := 2.220678;
   B_f[4] := -1.25157;
   B_f[5] := 4.578326;
   B_f[6] := 2.17674;
   B_f[7] := 2.244341;
   B_f[8] := 1.866234;
   B_f[9] := 3.735034;
   B_f[10] := 3.467353;
   B_f[11] := 3.067147;
   B_f[12] := 1.449147;
   B_f[13] := 2.446681;
   B_f[14] := 2.289465;
   B_f[15] := 2.636452;
   B_g[0] := 0.3080097;
   B_g[1] := -0.9424474;
   B_g[2] := 1.189431;
   B_g[3] := 0.5203503;
   B_g[4] := 0.4323277;
   B_g[5] := 0.2964829;
   B_g[6] := 0.2804947;
   B_g[7] := 0.4193809;
   B_g[8] := -0.2291173;
   B_g[9] := -0.6056316;
   B_g[10] := 0.1097276;
   B_g[11] := 0.5897712;
   B_g[12] := -1.135963;
   B_g[13] := 0.01335022;
   B_g[14] := 0.4513035;
   B_g[15] := 0.2196934;
   B_o[0] := 2.335754;
   B_o[1] := 3.887475;
   B_o[2] := 2.626467;
   B_o[3] := 2.155241;
   B_o[4] := 2.649906;
   B_o[5] := 4.28426;
   B_o[6] := 4.14954;
   B_o[7] := 3.200745;
   B_o[8] := 5.45463;
   B_o[9] := 3.353262;
   B_o[10] := 3.323039;
   B_o[11] := 2.977836;
   B_o[12] := 1.728129;
   B_o[13] := 3.911216;
   B_o[14] := 3.44036;
   B_o[15] := 2.920467;
   FC_W[0,0] := 0.7669169;
   FC_W[0,1] := 1.543509;
   FC_W[0,2] := -0.2084425;
   FC_W[0,3] := 0.3831763;
   FC_W[0,4] := 0.7583044;
   FC_W[0,5] := 1.109857;
   FC_W[0,6] := -0.9595311;
   FC_W[0,7] := 1.223664;
   FC_W[0,8] := -0.2153417;
   FC_W[0,9] := -3.007562;
   FC_W[0,10] := -0.08471649;
   FC_W[0,11] := 0.1802094;
   FC_W[0,12] := 0.5889047;
   FC_W[0,13] := -0.00262935;
   FC_W[0,14] := -0.6058581;
   FC_W[0,15] := 1.842039;
   FC_W[1,0] := -0.8487685;
   FC_W[1,1] := -0.9250219;
   FC_W[1,2] := 0.9445646;
   FC_W[1,3] := -1.085958;
   FC_W[1,4] := -0.5253252;
   FC_W[1,5] := 1.28364;
   FC_W[1,6] := -2.581259;
   FC_W[1,7] := -2.11015;
   FC_W[1,8] := -0.2588663;
   FC_W[1,9] := -1.638881;
   FC_W[1,10] := 0.7625059;
   FC_W[1,11] := 0.1852254;
   FC_W[1,12] := 1.451144;
   FC_W[1,13] := -0.8299196;
   FC_W[1,14] := 1.545634;
   FC_W[1,15] := -2.185032;
   FC_W[2,0] := 0.7475959;
   FC_W[2,1] := 1.504202;
   FC_W[2,2] := -0.1312031;
   FC_W[2,3] := 0.3657818;
   FC_W[2,4] := 0.7630855;
   FC_W[2,5] := 1.201591;
   FC_W[2,6] := -1.162883;
   FC_W[2,7] := 1.290929;
   FC_W[2,8] := -0.2123444;
   FC_W[2,9] := -3.140102;
   FC_W[2,10] := -0.1087691;
   FC_W[2,11] := 0.1746952;
   FC_W[2,12] := 0.7010824;
   FC_W[2,13] := 0.01334399;
   FC_W[2,14] := -0.7500849;
   FC_W[2,15] := 1.867126;
   FC_W[3,0] := -0.4515257;
   FC_W[3,1] := 0.2679058;
   FC_W[3,2] := -0.3569754;
   FC_W[3,3] := -0.427686;
   FC_W[3,4] := -0.1579306;
   FC_W[3,5] := -0.3923714;
   FC_W[3,6] := 1.284722;
   FC_W[3,7] := -0.3958135;
   FC_W[3,8] := -0.6324036;
   FC_W[3,9] := -1.887968;
   FC_W[3,10] := 0.01953238;
   FC_W[3,11] := 0.6071926;
   FC_W[3,12] := -0.00418234;
   FC_W[3,13] := 1.141586;
   FC_W[3,14] := -0.5711394;
   FC_W[3,15] := -0.2558074;
   FC_W[4,0] := 1.293448;
   FC_W[4,1] := -0.1032543;
   FC_W[4,2] := 0.5750578;
   FC_W[4,3] := -1.996473;
   FC_W[4,4] := -0.4809738;
   FC_W[4,5] := -0.8753579;
   FC_W[4,6] := 0.7629985;
   FC_W[4,7] := -0.3190035;
   FC_W[4,8] := 0.4359301;
   FC_W[4,9] := 0.3454917;
   FC_W[4,10] := 0.01366996;
   FC_W[4,11] := 1.019565;
   FC_W[4,12] := -0.6115221;
   FC_W[4,13] := -1.562433;
   FC_W[4,14] := -1.108395;
   FC_W[4,15] := 1.566593;
   FC_W[5,0] := 0.4117669;
   FC_W[5,1] := -1.244087;
   FC_W[5,2] := 0.4808592;
   FC_W[5,3] := 1.402493;
   FC_W[5,4] := -0.05570108;
   FC_W[5,5] := -6.805983;
   FC_W[5,6] := -0.6967741;
   FC_W[5,7] := 0.7403681;
   FC_W[5,8] := 1.617177;
   FC_W[5,9] := -0.05372217;
   FC_W[5,10] := -1.226606;
   FC_W[5,11] := 0.2559492;
   FC_W[5,12] := 0.2326207;
   FC_W[5,13] := -0.5059701;
   FC_W[5,14] := 0.233328;
   FC_W[5,15] := -0.6140623;
   FC_W[6,0] := 0.6124878;
   FC_W[6,1] := 1.539171;
   FC_W[6,2] := -0.01028113;
   FC_W[6,3] := 0.6690703;
   FC_W[6,4] := -0.1426041;
   FC_W[6,5] := -1.263851;
   FC_W[6,6] := -0.3345167;
   FC_W[6,7] := 0.3387654;
   FC_W[6,8] := 0.4775158;
   FC_W[6,9] := 0.9633071;
   FC_W[6,10] := -0.1772437;
   FC_W[6,11] := 2.243752;
   FC_W[6,12] := -0.4048626;
   FC_W[6,13] := 0.6561325;
   FC_W[6,14] := -0.4484591;
   FC_W[6,15] := -0.6827317;
   FC_W[7,0] := -0.4402839;
   FC_W[7,1] := 0.2908818;
   FC_W[7,2] := -0.3820719;
   FC_W[7,3] := -0.4177974;
   FC_W[7,4] := -0.1748291;
   FC_W[7,5] := -0.4283756;
   FC_W[7,6] := 1.368432;
   FC_W[7,7] := -0.3904219;
   FC_W[7,8] := -0.6243094;
   FC_W[7,9] := -1.802419;
   FC_W[7,10] := 0.04712024;
   FC_W[7,11] := 0.6073067;
   FC_W[7,12] := -0.07031967;
   FC_W[7,13] := 1.142984;
   FC_W[7,14] := -0.5244644;
   FC_W[7,15] := -0.2512715;
   FC_W[8,0] := -0.5053339;
   FC_W[8,1] := 0.3055462;
   FC_W[8,2] := -0.3846416;
   FC_W[8,3] := -0.4850571;
   FC_W[8,4] := -0.07984031;
   FC_W[8,5] := -0.3582116;
   FC_W[8,6] := 1.202516;
   FC_W[8,7] := -0.4420547;
   FC_W[8,8] := -0.6495288;
   FC_W[8,9] := -2.030459;
   FC_W[8,10] := 0.04362446;
   FC_W[8,11] := 0.5958719;
   FC_W[8,12] := 0.1207976;
   FC_W[8,13] := 1.117981;
   FC_W[8,14] := -0.6335613;
   FC_W[8,15] := -0.2960421;
   FC_W[9,0] := -0.4508871;
   FC_W[9,1] := 0.2760286;
   FC_W[9,2] := -0.3735214;
   FC_W[9,3] := -0.4126391;
   FC_W[9,4] := -0.1606828;
   FC_W[9,5] := -0.4006178;
   FC_W[9,6] := 1.317668;
   FC_W[9,7] := -0.3822564;
   FC_W[9,8] := -0.6318758;
   FC_W[9,9] := -1.855952;
   FC_W[9,10] := 0.04726556;
   FC_W[9,11] := 0.5970709;
   FC_W[9,12] := -0.0267396;
   FC_W[9,13] := 1.143159;
   FC_W[9,14] := -0.5352381;
   FC_W[9,15] := -0.252293;
   FC_W[10,0] := -1.112556;
   FC_W[10,1] := -1.107588;
   FC_W[10,2] := -0.2471485;
   FC_W[10,3] := -0.5994098;
   FC_W[10,4] := -0.1081943;
   FC_W[10,5] := -1.587787;
   FC_W[10,6] := 0.6018096;
   FC_W[10,7] := -0.6966217;
   FC_W[10,8] := -0.6367503;
   FC_W[10,9] := -3.216729;
   FC_W[10,10] := 0.03261364;
   FC_W[10,11] := -1.075626;
   FC_W[10,12] := 0.9282531;
   FC_W[10,13] := 0.363622;
   FC_W[10,14] := 0.1423627;
   FC_W[10,15] := -0.2397637;
   FC_W[11,0] := -0.03737991;
   FC_W[11,1] := -0.06299526;
   FC_W[11,2] := 0.6195287;
   FC_W[11,3] := 0.1934192;
   FC_W[11,4] := -1.420157;
   FC_W[11,5] := 0.08432721;
   FC_W[11,6] := 0.3095265;
   FC_W[11,7] := 0.8113614;
   FC_W[11,8] := -1.678368;
   FC_W[11,9] := -0.01523663;
   FC_W[11,10] := -0.8719974;
   FC_W[11,11] := 0.1192229;
   FC_W[11,12] := 0.3813153;
   FC_W[11,13] := -0.287847;
   FC_W[11,14] := -0.1337761;
   FC_W[11,15] := -0.1166494;
   FC_W[12,0] := -0.2101358;
   FC_W[12,1] := -0.2508407;
   FC_W[12,2] := 0.699504;
   FC_W[12,3] := 0.1080372;
   FC_W[12,4] := -1.519415;
   FC_W[12,5] := 0.05514818;
   FC_W[12,6] := -0.01964889;
   FC_W[12,7] := 1.257296;
   FC_W[12,8] := -1.133591;
   FC_W[12,9] := -0.04563072;
   FC_W[12,10] := -0.3616004;
   FC_W[12,11] := -0.04378428;
   FC_W[12,12] := 0.1271594;
   FC_W[12,13] := -0.02202382;
   FC_W[12,14] := -0.2301139;
   FC_W[12,15] := -0.3006166;
   FC_W[13,0] := 0.7408952;
   FC_W[13,1] := -0.07237465;
   FC_W[13,2] := 0.01080942;
   FC_W[13,3] := -0.1376049;
   FC_W[13,4] := -0.403186;
   FC_W[13,5] := 0.09405857;
   FC_W[13,6] := -0.6244625;
   FC_W[13,7] := 0.107715;
   FC_W[13,8] := -0.5213009;
   FC_W[13,9] := -0.5592325;
   FC_W[13,10] := 2.080232;
   FC_W[13,11] := -0.2632575;
   FC_W[13,12] := -0.6006549;
   FC_W[13,13] := 0.7337074;
   FC_W[13,14] := 4.43074;
   FC_W[13,15] := -1.039708;
   FC_W[14,0] := -3.11081;
   FC_W[14,1] := 1.525147;
   FC_W[14,2] := -0.3000883;
   FC_W[14,3] := -3.753221;
   FC_W[14,4] := 0.6175813;
   FC_W[14,5] := 0.7986314;
   FC_W[14,6] := 0.8566551;
   FC_W[14,7] := 2.646843;
   FC_W[14,8] := 1.932088;
   FC_W[14,9] := -0.0278612;
   FC_W[14,10] := -3.762145;
   FC_W[14,11] := 2.244887;
   FC_W[14,12] := 2.171723;
   FC_W[14,13] := 0.5284947;
   FC_W[14,14] := 2.066213;
   FC_W[14,15] := 0.2130263;
   FC_W[15,0] := 0.1661606;
   FC_W[15,1] := 0.1062202;
   FC_W[15,2] := 0.533263;
   FC_W[15,3] := 0.3180712;
   FC_W[15,4] := -1.174404;
   FC_W[15,5] := 0.08476182;
   FC_W[15,6] := 0.1170504;
   FC_W[15,7] := -0.01000034;
   FC_W[15,8] := -2.36727;
   FC_W[15,9] := 0.03094;
   FC_W[15,10] := -1.626169;
   FC_W[15,11] := 0.3396509;
   FC_W[15,12] := 0.6075796;
   FC_W[15,13] := -0.1496591;
   FC_W[15,14] := -0.00611463;
   FC_W[15,15] := 0.407406;
   FC_W[16,0] := -0.9638089;
   FC_W[16,1] := 1.081688;
   FC_W[16,2] := 2.376685;
   FC_W[16,3] := -1.057313;
   FC_W[16,4] := 0.292491;
   FC_W[16,5] := -0.3691578;
   FC_W[16,6] := -3.404121;
   FC_W[16,7] := -3.52346;
   FC_W[16,8] := -0.0705777;
   FC_W[16,9] := 0.6342216;
   FC_W[16,10] := -1.44417;
   FC_W[16,11] := -0.8829482;
   FC_W[16,12] := 0.7455462;
   FC_W[16,13] := 4.628078;
   FC_W[16,14] := 0.4031379;
   FC_W[16,15] := 3.93857;
   FC_W[17,0] := -1.180362;
   FC_W[17,1] := -0.2854657;
   FC_W[17,2] := 1.83997;
   FC_W[17,3] := -0.8665327;
   FC_W[17,4] := -0.6279789;
   FC_W[17,5] := -0.241897;
   FC_W[17,6] := -1.593776;
   FC_W[17,7] := 3.173894;
   FC_W[17,8] := 4.203144;
   FC_W[17,9] := 0.3790003;
   FC_W[17,10] := 3.867665;
   FC_W[17,11] := -2.212742;
   FC_W[17,12] := -1.379584;
   FC_W[17,13] := 1.736728;
   FC_W[17,14] := -0.7169582;
   FC_W[17,15] := -1.048066;
   FC_W[18,0] := 0.1636339;
   FC_W[18,1] := 2.465247;
   FC_W[18,2] := -0.7892377;
   FC_W[18,3] := 0.8747643;
   FC_W[18,4] := -5.954097;
   FC_W[18,5] := 0.8895477;
   FC_W[18,6] := 1.853717;
   FC_W[18,7] := -0.909115;
   FC_W[18,8] := 1.678992;
   FC_W[18,9] := 0.08326869;
   FC_W[18,10] := -0.3331011;
   FC_W[18,11] := -1.379958;
   FC_W[18,12] := 0.1766867;
   FC_W[18,13] := -1.740944;
   FC_W[18,14] := -0.1467744;
   FC_W[18,15] := 0.7952656;
   FC_W[19,0] := -0.2545704;
   FC_W[19,1] := -0.9416297;
   FC_W[19,2] := 0.5701975;
   FC_W[19,3] := -0.06669754;
   FC_W[19,4] := -0.3189588;
   FC_W[19,5] := -0.1196937;
   FC_W[19,6] := -0.3763052;
   FC_W[19,7] := 1.847393;
   FC_W[19,8] := -1.244459;
   FC_W[19,9] := -0.0925235;
   FC_W[19,10] := -0.06256182;
   FC_W[19,11] := 0.3304904;
   FC_W[19,12] := -0.05521645;
   FC_W[19,13] := 0.08963338;
   FC_W[19,14] := -0.2452032;
   FC_W[19,15] := -0.763625;
   FC_W[20,0] := -0.4479448;
   FC_W[20,1] := -2.149608;
   FC_W[20,2] := 0.2959174;
   FC_W[20,3] := -0.1774364;
   FC_W[20,4] := -0.5836748;
   FC_W[20,5] := 0.5884709;
   FC_W[20,6] := 1.354637;
   FC_W[20,7] := -0.1612765;
   FC_W[20,8] := -0.2719716;
   FC_W[20,9] := -0.6377214;
   FC_W[20,10] := 0.5176937;
   FC_W[20,11] := -1.327186;
   FC_W[20,12] := 0.3548906;
   FC_W[20,13] := -0.7838172;
   FC_W[20,14] := 0.8982322;
   FC_W[20,15] := 1.425032;
   FC_W[21,0] := -2.43107;
   FC_W[21,1] := 1.030155;
   FC_W[21,2] := -0.236344;
   FC_W[21,3] := 1.300441;
   FC_W[21,4] := 0.4406562;
   FC_W[21,5] := 0.7007543;
   FC_W[21,6] := -0.385313;
   FC_W[21,7] := 0.1291319;
   FC_W[21,8] := -0.4665849;
   FC_W[21,9] := -0.6554801;
   FC_W[21,10] := 0.3629912;
   FC_W[21,11] := 1.437753;
   FC_W[21,12] := -0.3645638;
   FC_W[21,13] := -0.4504355;
   FC_W[21,14] := -0.5624921;
   FC_W[21,15] := 1.265119;
   FC_W[22,0] := 0.2240193;
   FC_W[22,1] := -1.527885;
   FC_W[22,2] := 2.091162;
   FC_W[22,3] := 0.5646194;
   FC_W[22,4] := -0.4624339;
   FC_W[22,5] := 0.7368477;
   FC_W[22,6] := 0.1916436;
   FC_W[22,7] := 0.06346934;
   FC_W[22,8] := 0.5419989;
   FC_W[22,9] := -1.039653;
   FC_W[22,10] := -0.2493821;
   FC_W[22,11] := 2.156514;
   FC_W[22,12] := -1.799162;
   FC_W[22,13] := -0.2155053;
   FC_W[22,14] := 0.6050608;
   FC_W[22,15] := 0.5826755;
   FC_W[23,0] := 0.9354936;
   FC_W[23,1] := -0.4059404;
   FC_W[23,2] := -0.1648392;
   FC_W[23,3] := 0.02804452;
   FC_W[23,4] := -0.5441927;
   FC_W[23,5] := -0.1005955;
   FC_W[23,6] := 0.5784212;
   FC_W[23,7] := -0.1252794;
   FC_W[23,8] := -0.7804069;
   FC_W[23,9] := -0.6183712;
   FC_W[23,10] := 1.441071;
   FC_W[23,11] := -0.1692511;
   FC_W[23,12] := -0.8358346;
   FC_W[23,13] := 1.602945;
   FC_W[23,14] := 4.239077;
   FC_W[23,15] := -1.320831;
   FC_W[24,0] := 0.1837721;
   FC_W[24,1] := -1.394907;
   FC_W[24,2] := 1.99884;
   FC_W[24,3] := 0.550393;
   FC_W[24,4] := -0.580985;
   FC_W[24,5] := 0.6370355;
   FC_W[24,6] := 0.2918367;
   FC_W[24,7] := 0.03679674;
   FC_W[24,8] := 0.5497574;
   FC_W[24,9] := -0.8343722;
   FC_W[24,10] := -0.2216339;
   FC_W[24,11] := 2.071422;
   FC_W[24,12] := -2.016426;
   FC_W[24,13] := -0.236861;
   FC_W[24,14] := 0.7079917;
   FC_W[24,15] := 0.5801944;
   FC_W[25,0] := 0.1875129;
   FC_W[25,1] := -1.401109;
   FC_W[25,2] := 2.012083;
   FC_W[25,3] := 0.5548877;
   FC_W[25,4] := -0.5858603;
   FC_W[25,5] := 0.6392438;
   FC_W[25,6] := 0.2960918;
   FC_W[25,7] := 0.03836685;
   FC_W[25,8] := 0.5552443;
   FC_W[25,9] := -0.8309537;
   FC_W[25,10] := -0.2237335;
   FC_W[25,11] := 2.081445;
   FC_W[25,12] := -2.024895;
   FC_W[25,13] := -0.2364689;
   FC_W[25,14] := 0.7084617;
   FC_W[25,15] := 0.5862992;
   FC_W[26,0] := 1.663001;
   FC_W[26,1] := -1.822266;
   FC_W[26,2] := 1.667857;
   FC_W[26,3] := -0.6290205;
   FC_W[26,4] := 0.321302;
   FC_W[26,5] := -0.1651625;
   FC_W[26,6] := -0.3183419;
   FC_W[26,7] := -0.01305876;
   FC_W[26,8] := 0.2468822;
   FC_W[26,9] := -0.6432862;
   FC_W[26,10] := -0.01610377;
   FC_W[26,11] := 1.134091;
   FC_W[26,12] := -0.7709256;
   FC_W[26,13] := 0.5913879;
   FC_W[26,14] := 1.184353;
   FC_W[26,15] := -0.7892672;
   FC_W[27,0] := -2.892142;
   FC_W[27,1] := 1.406102;
   FC_W[27,2] := -0.8661692;
   FC_W[27,3] := 0.7728196;
   FC_W[27,4] := 0.7940138;
   FC_W[27,5] := 0.3448563;
   FC_W[27,6] := -0.3961662;
   FC_W[27,7] := -0.09319982;
   FC_W[27,8] := -0.9166206;
   FC_W[27,9] := -0.4265728;
   FC_W[27,10] := 0.8124349;
   FC_W[27,11] := 0.8865057;
   FC_W[27,12] := -0.4073323;
   FC_W[27,13] := -0.5555975;
   FC_W[27,14] := -0.2353146;
   FC_W[27,15] := 1.349715;
   FC_W[28,0] := 1.562958;
   FC_W[28,1] := 1.421223;
   FC_W[28,2] := 0.00074465;
   FC_W[28,3] := -2.077267;
   FC_W[28,4] := 0.4371008;
   FC_W[28,5] := -1.419437;
   FC_W[28,6] := -0.5331396;
   FC_W[28,7] := -0.04702906;
   FC_W[28,8] := -0.3670209;
   FC_W[28,9] := 0.3774387;
   FC_W[28,10] := 0.5960436;
   FC_W[28,11] := 2.106222;
   FC_W[28,12] := 0.02389226;
   FC_W[28,13] := -0.8460939;
   FC_W[28,14] := -0.4706507;
   FC_W[28,15] := 0.4614136;
   FC_W[29,0] := 0.1833606;
   FC_W[29,1] := 1.359581;
   FC_W[29,2] := -1.921257;
   FC_W[29,3] := -0.4466536;
   FC_W[29,4] := 0.6786666;
   FC_W[29,5] := -1.270405;
   FC_W[29,6] := 0.3430922;
   FC_W[29,7] := 0.3040659;
   FC_W[29,8] := -0.2850345;
   FC_W[29,9] := 2.146905;
   FC_W[29,10] := -0.1342847;
   FC_W[29,11] := -2.2644;
   FC_W[29,12] := 0.5790378;
   FC_W[29,13] := 0.4808839;
   FC_W[29,14] := -0.5187714;
   FC_W[29,15] := -0.6746457;
   FC_W[30,0] := 0.2279541;
   FC_W[30,1] := -1.531598;
   FC_W[30,2] := 2.093725;
   FC_W[30,3] := 0.5648265;
   FC_W[30,4] := -0.4606146;
   FC_W[30,5] := 0.7382425;
   FC_W[30,6] := 0.1888482;
   FC_W[30,7] := 0.06514335;
   FC_W[30,8] := 0.5416202;
   FC_W[30,9] := -1.043393;
   FC_W[30,10] := -0.2514903;
   FC_W[30,11] := 2.156712;
   FC_W[30,12] := -1.79456;
   FC_W[30,13] := -0.2139972;
   FC_W[30,14] := 0.6010243;
   FC_W[30,15] := 0.58391;
   FC_W[31,0] := 0.2782316;
   FC_W[31,1] := -1.584971;
   FC_W[31,2] := 2.129416;
   FC_W[31,3] := 0.5732425;
   FC_W[31,4] := -0.4093653;
   FC_W[31,5] := 0.7742324;
   FC_W[31,6] := 0.1738364;
   FC_W[31,7] := 0.1063647;
   FC_W[31,8] := 0.5556461;
   FC_W[31,9] := -1.073487;
   FC_W[31,10] := -0.2855354;
   FC_W[31,11] := 2.192433;
   FC_W[31,12] := -1.709227;
   FC_W[31,13] := -0.1924735;
   FC_W[31,14] := 0.529599;
   FC_W[31,15] := 0.5927989;
   FC_W[32,0] := 0.04953038;
   FC_W[32,1] := -1.415494;
   FC_W[32,2] := 2.016365;
   FC_W[32,3] := 0.5011491;
   FC_W[32,4] := -0.4617985;
   FC_W[32,5] := 0.7487798;
   FC_W[32,6] := 0.134348;
   FC_W[32,7] := -0.03319941;
   FC_W[32,8] := 0.4558607;
   FC_W[32,9] := -1.141186;
   FC_W[32,10] := -0.1354079;
   FC_W[32,11] := 2.234947;
   FC_W[32,12] := -1.731302;
   FC_W[32,13] := -0.3103259;
   FC_W[32,14] := 0.6360376;
   FC_W[32,15] := 0.6504694;
   FC_W[33,0] := -0.00627907;
   FC_W[33,1] := -1.499087;
   FC_W[33,2] := 2.072517;
   FC_W[33,3] := 0.4723728;
   FC_W[33,4] := -0.2860313;
   FC_W[33,5] := 0.8612234;
   FC_W[33,6] := -0.05305826;
   FC_W[33,7] := -0.05858019;
   FC_W[33,8] := 0.4062904;
   FC_W[33,9] := -1.418352;
   FC_W[33,10] := -0.1284464;
   FC_W[33,11] := 2.384624;
   FC_W[33,12] := -1.412978;
   FC_W[33,13] := -0.3630248;
   FC_W[33,14] := 0.4452505;
   FC_W[33,15] := 0.6962806;
   FC_W[34,0] := 0.08176677;
   FC_W[34,1] := -1.524861;
   FC_W[34,2] := 2.100555;
   FC_W[34,3] := 0.5096552;
   FC_W[34,4] := -0.3558632;
   FC_W[34,5] := 0.8747145;
   FC_W[34,6] := 0.00432379;
   FC_W[34,7] := -0.01442015;
   FC_W[34,8] := 0.4600074;
   FC_W[34,9] := -1.383607;
   FC_W[34,10] := -0.1860707;
   FC_W[34,11] := 2.33854;
   FC_W[34,12] := -1.441226;
   FC_W[34,13] := -0.3380259;
   FC_W[34,14] := 0.4379412;
   FC_W[34,15] := 0.6816462;
   FC_W[35,0] := 0.0051369;
   FC_W[35,1] := -1.328843;
   FC_W[35,2] := 1.909314;
   FC_W[35,3] := 0.4985209;
   FC_W[35,4] := -0.5634329;
   FC_W[35,5] := 0.678765;
   FC_W[35,6] := 0.2334343;
   FC_W[35,7] := -0.06241892;
   FC_W[35,8] := 0.4209301;
   FC_W[35,9] := -1.01738;
   FC_W[35,10] := -0.03109938;
   FC_W[35,11] := 2.153967;
   FC_W[35,12] := -1.840335;
   FC_W[35,13] := -0.294865;
   FC_W[35,14] := 0.8384414;
   FC_W[35,15] := 0.6365836;
   FC_W[36,0] := -1.568046;
   FC_W[36,1] := 1.120774;
   FC_W[36,2] := 0.2148976;
   FC_W[36,3] := -0.856096;
   FC_W[36,4] := 0.4192909;
   FC_W[36,5] := -0.7212552;
   FC_W[36,6] := -0.2086197;
   FC_W[36,7] := -0.4754252;
   FC_W[36,8] := 0.0581672;
   FC_W[36,9] := 0.8853021;
   FC_W[36,10] := -1.338137;
   FC_W[36,11] := -1.436484;
   FC_W[36,12] := -6.047898;
   FC_W[36,13] := -0.4120009;
   FC_W[36,14] := 0.4727429;
   FC_W[36,15] := -0.3096007;
   FC_W[37,0] := -0.01744911;
   FC_W[37,1] := -1.288111;
   FC_W[37,2] := 1.874067;
   FC_W[37,3] := 0.493008;
   FC_W[37,4] := -0.576397;
   FC_W[37,5] := 0.6525027;
   FC_W[37,6] := 0.2459292;
   FC_W[37,7] := -0.07283052;
   FC_W[37,8] := 0.4050449;
   FC_W[37,9] := -0.9737098;
   FC_W[37,10] := -0.00745488;
   FC_W[37,11] := 2.125903;
   FC_W[37,12] := -1.89184;
   FC_W[37,13] := -0.2835879;
   FC_W[37,14] := 0.8971778;
   FC_W[37,15] := 0.617029;
   FC_W[38,0] := -0.2852966;
   FC_W[38,1] := -2.812381;
   FC_W[38,2] := -3.517689;
   FC_W[38,3] := 0.4010945;
   FC_W[38,4] := -0.9821432;
   FC_W[38,5] := 0.3339402;
   FC_W[38,6] := -3.252781;
   FC_W[38,7] := -1.330081;
   FC_W[38,8] := 0.2798223;
   FC_W[38,9] := -1.038314;
   FC_W[38,10] := 0.04537877;
   FC_W[38,11] := 2.10163;
   FC_W[38,12] := -1.06387;
   FC_W[38,13] := 1.874116;
   FC_W[38,14] := -0.5416867;
   FC_W[38,15] := 1.843496;
   FC_W[39,0] := -1.929015;
   FC_W[39,1] := -0.7853311;
   FC_W[39,2] := -2.235025;
   FC_W[39,3] := -1.940823;
   FC_W[39,4] := -0.1226789;
   FC_W[39,5] := 0.6661553;
   FC_W[39,6] := -1.054318;
   FC_W[39,7] := 1.030784;
   FC_W[39,8] := 1.43678;
   FC_W[39,9] := -0.6748919;
   FC_W[39,10] := -2.097334;
   FC_W[39,11] := 2.614807;
   FC_W[39,12] := 0.5899004;
   FC_W[39,13] := 1.10489;
   FC_W[39,14] := 0.7451716;
   FC_W[39,15] := 0.8715423;
   FC_B[0] := -0.333644;
   FC_B[1] := -0.07630836;
   FC_B[2] := -0.3470396;
   FC_B[3] := 0.05934331;
   FC_B[4] := -0.6669545;
   FC_B[5] := -0.1396796;
   FC_B[6] := 0.4899451;
   FC_B[7] := 0.06493863;
   FC_B[8] := 0.09218118;
   FC_B[9] := 0.06467691;
   FC_B[10] := -0.1966108;
   FC_B[11] := -0.4983726;
   FC_B[12] := -0.4815665;
   FC_B[13] := -0.839667;
   FC_B[14] := 0.7280124;
   FC_B[15] := -0.5059478;
   FC_B[16] := 0.144936;
   FC_B[17] := 0.02873158;
   FC_B[18] := 1.814771;
   FC_B[19] := -0.8144414;
   FC_B[20] := -0.8217906;
   FC_B[21] := 0.4051378;
   FC_B[22] := -1.708364;
   FC_B[23] := -0.887781;
   FC_B[24] := -1.654905;
   FC_B[25] := -1.662859;
   FC_B[26] := -1.66001;
   FC_B[27] := 0.6486168;
   FC_B[28] := -0.2243079;
   FC_B[29] := 1.429813;
   FC_B[30] := -1.709721;
   FC_B[31] := -1.722916;
   FC_B[32] := -1.654223;
   FC_B[33] := -1.667235;
   FC_B[34] := -1.678131;
   FC_B[35] := -1.616012;
   FC_B[36] := -0.6812373;
   FC_B[37] := -1.60075;
   FC_B[38] := 0.8395569;
   FC_B[39] := 0.8761413;

END_DATA_BLOCK

FUNCTION "_RestartTesting" : Int
{ S7_Optimized_Access := 'TRUE' }
VERSION : 0.1
   VAR_INPUT
      bStart : Bool;
   END_VAR


BEGIN
	IF #bStart THEN
	    "DB_Main".PredictCount := 0;
	    "DB_Result".TruePositive := 0;
	    "DB_Result".TrueNegative := 0;
	    "DB_Result".FalsePositive := 0;
	    "DB_Result".FalseNegative := 0;
	    #_RestartTesting := 10;
	ELSE
	    #_RestartTesting := 0;
	END_IF;
END_FUNCTION

FUNCTION "_Zscore" : Real
{ S7_Optimized_Access := 'TRUE' }
VERSION : 0.1
   VAR_INPUT
      iRow : Int;
      iCol : Int;
   END_VAR


BEGIN
	#_Zscore := ("DB_Attack_v0_first_attack".DATA[#iRow, #iCol] - "DB_FeatureNormRef_Means".Means[#iCol]) / "DB_FeatureNormRef_std".std[#iCol];

END_FUNCTION

FUNCTION "_LIMIT" : Real
{ S7_Optimized_Access := 'TRUE' }
VERSION : 0.1
   VAR_INPUT
      inVal : Real;
      minVal : Real;
      maxVal : Real;
   END_VAR

   VAR_TEMP
      lo : Real;
      hi : Real;
   END_VAR


BEGIN
	IF #inVal < #minVal THEN
	    #_LIMIT := #minVal;
	ELSIF #inVal > #maxVal THEN
	    #_LIMIT := #maxVal;
	ELSE
	    #_LIMIT := #inVal;
	END_IF;

END_FUNCTION

FUNCTION "_FC_layer" : Void
{ S7_Optimized_Access := 'TRUE' }
VERSION : 0.1
   VAR_INPUT
      h_t : Array[0..15] of Real;
   END_VAR

   VAR_OUTPUT
      y : Array[0..39] of Real;
   END_VAR

   VAR_TEMP
      i : Int;
      j : Int;
   END_VAR


BEGIN
	FOR #i := 0 TO 39 DO
	    #y[#i] := 0.0;
	    FOR #j := 0 TO 15 DO
	        #y[#i] := #y[#i] + "DB_model_HS16_IW10".FC_W[#i, #j] * #h_t[#j];
	    END_FOR;
	    #y[#i] := #y[#i] + "DB_model_HS16_IW10".FC_B[#i];
	END_FOR;
END_FUNCTION

DATA_BLOCK "DB_Measuring"
{ S7_Optimized_Access := 'TRUE' }
VERSION : 0.1
NON_RETAIN
   VAR
      CycleTime_ms : DInt;
      last_cycle_time : LTime;
      last_cycle_ms : Array[0..3000] of DInt;
   END_VAR


BEGIN

END_DATA_BLOCK

DATA_BLOCK "DB_LSTM"
{ S7_Optimized_Access := 'TRUE' }
VERSION : 0.1
NON_RETAIN
   VAR
      c_tm1 : Array[0..15] of Real;
      h_tm1 : Array[0..15] of Real;
      x_t : Array[0..99, 0..39] of Real;
      c_t : Array[0..15] of Real;
      h_t : Array[0..15] of Real;
      y : Array[0..39] of Real;
   END_VAR


BEGIN

END_DATA_BLOCK

ORGANIZATION_BLOCK "Main"
TITLE = "Main Program Sweep (Cycle)"
{ S7_Optimized_Access := 'TRUE' }
VERSION : 0.1
   VAR_TEMP
      f_t : Array[0..15] of Real;
      g_t : Array[0..15] of Real;
      o_t : Array[0..15] of Real;
      x_ct : Real;
      x_o : Real;
      x_g : Real;
      i_t : Array[0..15] of Real;
      x_f : Real;
      x_i : Real;
      k : Int;
      t : Int;
      I : Int;
      j : Int;
      predicted_class : Int;
      lastCycleTime : DInt;
      vInfo : Variant;
      retVal : Int;
   END_VAR


BEGIN
	        //-->> Cycle Time measuring
	#retVal:= RT_INFO(
	                  MODE := 25,
	                  OB := 1,
	                  INFO := "DB_Measuring".last_cycle_time
	);
	"DB_Measuring".last_cycle_ms["DB_Main".PredictCount]:= LTIME_TO_DINT("DB_Measuring".last_cycle_time);
	"DB_Measuring".CycleTime_ms := LTIME_TO_DINT("DB_Measuring".last_cycle_time) /1000000;


	 CASE "DB_Main".iState OF
	        //-->> IDLE
	    0:
	        "DB_Main".iState := "_RestartTesting"("DB_Main".bStart);


	        //-->> Fill Model Window
	    10:
	        FOR #I := 0 TO 15 DO
	            "DB_LSTM".h_tm1[#I] := 0.0;
	            "DB_LSTM".c_tm1[#I] := 0.0;
	        END_FOR;

	        FOR #I := 0 TO 9 DO
	            FOR #j := 0 TO 39 DO
	                "DB_LSTM".x_t[#I, #j] := "_Zscore"(iRow := #I, iCol := #j);
	            END_FOR;
	        END_FOR;
	        "DB_Result".TrueNegative := 100;
	        "DB_Main".PredictCount := 100;
	        "DB_Main".iState := 20;


	        //-->> Call LSTM modell
	    20:
	        FOR #I := 0 TO 15 DO
	            "DB_LSTM".c_tm1[#I] := 0.0;
	            "DB_LSTM".h_tm1[#I] := 0.0;
	        END_FOR;

	        FOR #t := 0 TO 9 DO
	            FOR #I := 0 TO 15 DO

	                // ---- Input gate ----
	                #x_i := "DB_model_HS16_IW10".B_i[#I];
	                FOR #k := 0 TO 39 DO
	                    #x_i := #x_i
	                    + "DB_model_HS16_IW10".W_i[#I, #k]
	                    * "DB_LSTM".x_t[#t, #k];
	                END_FOR;
	                FOR #j := 0 TO 15 DO
	                    #x_i := #x_i
	                    + "DB_model_HS16_IW10".R_i[#I, #j]
	                    * "DB_LSTM".h_tm1[#j];
	                END_FOR;
	                #x_i := "_LIMIT"(inVal := #x_i, maxVal := 20, minVal := -20);
	                #i_t[#I] := 1.0 / (1.0 + EXP(- #x_i));

	                // ---- Forget gate ----
	                #x_f := "DB_model_HS16_IW10".B_f[#I];
	                FOR #k := 0 TO 39 DO
	                    #x_f := #x_f
	                    + "DB_model_HS16_IW10".W_f[#I, #k]
	                    * "DB_LSTM".x_t[#t, #k];
	                END_FOR;
	                FOR #j := 0 TO 15 DO
	                    #x_f := #x_f
	                    + "DB_model_HS16_IW10".R_f[#I, #j]
	                    * "DB_LSTM".h_tm1[#j];
	                END_FOR;
	                #x_f := "_LIMIT"(inVal := #x_f, maxVal := 20, minVal := -20);
	                #f_t[#I] := 1.0 / (1.0 + EXP(- #x_f));

	                // ---- Cell candidate (tanh) ----
	                #x_g := "DB_model_HS16_IW10".B_g[#I];
	                FOR #k := 0 TO 39 DO
	                    #x_g := #x_g
	                    + "DB_model_HS16_IW10".W_g[#I, #k]
	                    * "DB_LSTM".x_t[#t, #k];
	                END_FOR;
	                FOR #j := 0 TO 15 DO
	                    #x_g := #x_g
	                    + "DB_model_HS16_IW10".R_g[#I, #j]
	                    * "DB_LSTM".h_tm1[#j];
	                END_FOR;
	                #x_g := "_LIMIT"(inVal := #x_g, maxVal := 20, minVal := -20);
	                #g_t[#I] := (EXP(#x_g) - EXP(- #x_g)) / (EXP(#x_g) + EXP(- #x_g)); // tanh

	                // ---- Output gate (sigmoid) ----
	                #x_o := "DB_model_HS16_IW10".B_o[#I];
	                FOR #k := 0 TO 39 DO
	                    #x_o := #x_o
	                    + "DB_model_HS16_IW10".W_o[#I, #k]
	                    * "DB_LSTM".x_t[#t, #k];
	                END_FOR;
	                FOR #j := 0 TO 15 DO
	                    #x_o := #x_o
	                    + "DB_model_HS16_IW10".R_o[#I, #j]
	                    * "DB_LSTM".h_tm1[#j];
	                END_FOR;
	                #x_o := "_LIMIT"(inVal := #x_o, maxVal := 20, minVal := -20);
	                #o_t[#I] := 1.0 / (1.0 + EXP(- #x_o));

	                // ---- Cell state frissítés ----
	                "DB_LSTM".c_t[#I] := #f_t[#I] * "DB_LSTM".c_tm1[#I] + #i_t[#I] * #g_t[#I];

	                // ---- Hidden state (tanh) ----
	                #x_ct := "_LIMIT"(inVal := "DB_LSTM".c_t[#I], maxVal := 20, minVal := -20);
	                "DB_LSTM".h_t[#I] := #o_t[#I] * ((EXP(#x_ct) - EXP(- #x_ct)) / (EXP(#x_ct) + EXP(- #x_ct)));
	            END_FOR;

	            FOR #I := 0 TO 15 DO
	                "DB_LSTM".c_tm1[#I] := "DB_LSTM".c_t[#I];
	                "DB_LSTM".h_tm1[#I] := "DB_LSTM".h_t[#I];
	            END_FOR;
	        END_FOR;

	        // Fully connected layer
	        "_FC_layer"(h_t := "DB_LSTM".h_t,
	                    y => "DB_LSTM".y);

	        // MSE calculation
	        "DB_Main".Mse := 0.0;
	        FOR #k := 0 TO 39 DO
	            "DB_Main".Mse := "DB_Main".Mse
	            + ("DB_LSTM".x_t[9, #k] - "DB_LSTM".y[#k])
	            * ("DB_LSTM".x_t[9, #k] - "DB_LSTM".y[#k]);
	        END_FOR;
	        "DB_Main".Mse := "DB_Main".Mse / INT_TO_REAL(40);

	        // Attack / Normal decision
	        IF "DB_Main".Mse > "DB_Result".THRESHOLD THEN
	            #predicted_class := 1;  // Attack
	        ELSE
	            #predicted_class := 0;  // Normal
	        END_IF;
	        "DB_Result".Predicted_class := #predicted_class;

	        IF "DB_Result".Predicted_class = 1 AND
	            REAL_TO_INT("DB_Attack_v0_first_attack".DATA["DB_Main".PredictCount, 40]) = 1
	        THEN
	            "DB_Result".TruePositive := "DB_Result".TruePositive + 1;
	        ELSIF "DB_Result".Predicted_class = 0 AND
	            REAL_TO_INT("DB_Attack_v0_first_attack".DATA["DB_Main".PredictCount, 40]) = 0
	        THEN
	            "DB_Result".TrueNegative := "DB_Result".TrueNegative + 1;
	        ELSIF "DB_Result".Predicted_class = 1 AND
	            REAL_TO_INT("DB_Attack_v0_first_attack".DATA["DB_Main".PredictCount, 40]) = 0
	        THEN
	            "DB_Result".FalsePositive := "DB_Result".FalsePositive + 1;
	        ELSIF "DB_Result".Predicted_class = 0 AND
	            REAL_TO_INT("DB_Attack_v0_first_attack".DATA["DB_Main".PredictCount, 40]) = 1
	        THEN
	            "DB_Result".FalseNegative := "DB_Result".FalseNegative + 1;
	        END_IF;
	        "DB_Main".PredictCount := "DB_Main".PredictCount + 1;

	        IF "DB_Main".PredictCount >= "DB_Result".EXPECTED_PREDICITON_COUNT THEN
	            "DB_Main".iState  := 100;
	        ELSE

	            FOR #I := 0 TO 8 DO
	                FOR #j := 0 TO 39 DO
	                    "DB_LSTM".x_t[#I, #j] := "DB_LSTM".x_t[#I + 1, #j];
	                END_FOR;
	            END_FOR;

	            FOR #j := 0 TO 39 DO
	                "DB_LSTM".x_t[9, #j] := "_Zscore"(iRow := "DB_Main".PredictCount, iCol := #j);
	            END_FOR;
	            "DB_Main".iState := 20;
	        END_IF;


	        //-->> Test Ready Compare Result
	    100:
	        IF "DB_Result".TrueNegative <> "DB_Result".EXPECTED_TRUE_NEGATIVE THEN
	            "DB_Result".MismatchCount := "DB_Result".MismatchCount + 1;
	        END_IF;
	        IF "DB_Result".FalsePositive <>"DB_Result".EXPECTED_FALSE_POSITIVE THEN
	            "DB_Result".MismatchCount := "DB_Result".MismatchCount + 1;
	        END_IF;
	        IF "DB_Result".FalseNegative <> "DB_Result".EXPECTED_FALSE_NEGATIVE THEN
	            "DB_Result".MismatchCount := "DB_Result".MismatchCount + 1;
	        END_IF;
	        IF "DB_Result".TruePositive <> "DB_Result".EXPECTED_TRUE_POSITIVE THEN
	            "DB_Result".MismatchCount := "DB_Result".MismatchCount + 1;
	        END_IF;
	        IF "DB_Main".PredictCount <> "DB_Result".EXPECTED_PREDICITON_COUNT THEN
	            "DB_Result".MismatchCount := "DB_Result".MismatchCount + 1;
	        END_IF;
	        IF "DB_Result".MismatchCount <> 0 THEN
	            "DB_Main".iState := 150;
	        ELSE
	            "DB_Main".iState := 200;
	        END_IF;


	    150,200:
	        IF NOT "DB_Main".bStart THEN
	            "DB_Main".iState := 0;
	        END_IF;

	  END_CASE;
END_ORGANIZATION_BLOCK

